LIN {X 0,Y 523.933,Z 425.84,A -85,B 0,C 180,E1 -4843.639,E2 -4843.639} C_VEL
LIN {X 0,Y 523.933,Z 425.846,A -85,B 0,C 180,E1 -4846.028,E2 -4846.028} C_VEL
LIN {X 0,Y 524.007,Z 425.841,A -85,B 0,C 180,E1 -4848.394,E2 -4848.394} C_VEL
LIN {X 0,Y 524,Z 425.833,A -85,B 0,C 180,E1 -4851.516,E2 -4851.516} C_VEL
LIN {X 0,Y 524.077,Z 425.829,A -85,B 0,C 180,E1 -4854.614,E2 -4854.614} C_VEL
LIN {X 0,Y 524.106,Z 425.82,A -85,B 0,C 180,E1 -4857.695,E2 -4857.695} C_VEL
LIN {X 0,Y 524.118,Z 425.82,A -85,B 0,C 180,E1 -4860.769,E2 -4860.769} C_VEL
LIN {X 0,Y 524.069,Z 425.826,A -85,B 0,C 180,E1 -4863.075,E2 -4863.075} C_VEL
LIN {X 0,Y 524.045,Z 425.833,A -85,B 0,C 180,E1 -4866.159,E2 -4866.159} C_VEL
LIN {X 0,Y 523.996,Z 425.834,A -85,B 0,C 180,E1 -4869.262,E2 -4869.262} C_VEL
LIN {X 0,Y 523.996,Z 425.834,A -85,B 0,C 180,E1 -4871.74,E2 -4871.74} C_VEL
LIN {X 0,Y 523.987,Z 425.837,A -85,B 0,C 180,E1 -4875.053,E2 -4875.053} C_VEL
LIN {X 0,Y 523.958,Z 425.842,A -85,B 0,C 180,E1 -4877.969,E2 -4877.969} C_VEL
LIN {X 0,Y 523.966,Z 425.847,A -85,B 0,C 180,E1 -4880.411,E2 -4880.411} C_VEL
LIN {X 0,Y 523.911,Z 425.848,A -85,B 0,C 180,E1 -4882.894,E2 -4882.894} C_VEL
LIN {X 0,Y 523.949,Z 425.841,A -85,B 0,C 180,E1 -4885.419,E2 -4885.419} C_VEL
LIN {X 0,Y 523.966,Z 425.842,A -85,B 0,C 180,E1 -4887.999,E2 -4887.999} C_VEL
LIN {X 0,Y 523.948,Z 425.845,A -85,B 0,C 180,E1 -4890.857,E2 -4890.857} C_VEL
LIN {X 0,Y 523.958,Z 425.841,A -85,B 0,C 180,E1 -4893.736,E2 -4893.736} C_VEL
LIN {X 0,Y 523.921,Z 425.852,A -85,B 0,C 180,E1 -4896.406,E2 -4896.406} C_VEL
LIN {X 0,Y 523.956,Z 425.844,A -85,B 0,C 180,E1 -4899.082,E2 -4899.082} C_VEL
LIN {X 0,Y 523.953,Z 425.847,A -85,B 0,C 180,E1 -4902.119,E2 -4902.119} C_VEL
LIN {X 0,Y 524.002,Z 426.023,A -85,B 0,C 180,E1 -4903.252,E2 -4903.252} C_VEL
LIN {X 0,Y 525.992,Z 435.927,A -85,B 0,C 180,E1 -4904.916,E2 -4904.916} C_VEL
LIN {X 0,Y 525.874,Z 439.256,A -85,B 0,C 180,E1 -4905.427,E2 -4905.427} C_VEL
LIN {X 0,Y 525.617,Z 441.85,A -85,B 0,C 180,E1 -4905.741,E2 -4905.741} C_VEL
LIN {X 0,Y 524.85,Z 446.612,A -85,B 0,C 180,E1 -4906.106,E2 -4906.106} C_VEL
LIN {X 0,Y 523.874,Z 451.969,A -85,B 0,C 180,E1 -4906.359,E2 -4906.359} C_VEL
LIN {X 0,Y 522.61,Z 459.806,A -85,B 0,C 180,E1 -4906.576,E2 -4906.576} C_VEL
LIN {X 0,Y 521.99,Z 467.878,A -85,B 0,C 180,E1 -4906.711,E2 -4906.711} C_VEL
LIN {X 0,Y 520.915,Z 611.533,A -85,B 0,C 180,E1 -4908.76,E2 -4908.76} C_VEL
LIN {X 0,Y 520.597,Z 626.808,A -85,B 0,C 180,E1 -4909.129,E2 -4909.129} C_VEL
LIN {X 0,Y 520.217,Z 641.341,A -85,B 0,C 180,E1 -4909.639,E2 -4909.639} C_VEL
LIN {X 0,Y 519.75,Z 655.45,A -85,B 0,C 180,E1 -4910.291,E2 -4910.291} C_VEL
LIN {X 0,Y 519.293,Z 667.726,A -85,B 0,C 180,E1 -4911.001,E2 -4911.001} C_VEL
LIN {X 0,Y 518.8,Z 680.193,A -85,B 0,C 180,E1 -4911.873,E2 -4911.873} C_VEL
LIN {X 0,Y 518.29,Z 692.73,A -85,B 0,C 180,E1 -4912.931,E2 -4912.931} C_VEL
LIN {X 0,Y 517.723,Z 704.894,A -85,B 0,C 180,E1 -4914.169,E2 -4914.169} C_VEL
LIN {X 0,Y 517.327,Z 715.213,A -85,B 0,C 180,E1 -4915.43,E2 -4915.43} C_VEL
LIN {X 0,Y 516.961,Z 724.771,A -85,B 0,C 180,E1 -4916.826,E2 -4916.826} C_VEL
LIN {X 0,Y 516.71,Z 732.578,A -85,B 0,C 180,E1 -4918.194,E2 -4918.194} C_VEL
LIN {X 0,Y 516.51,Z 739.956,A -85,B 0,C 180,E1 -4919.773,E2 -4919.773} C_VEL
LIN {X 0,Y 516.361,Z 745.035,A -85,B 0,C 180,E1 -4921.108,E2 -4921.108} C_VEL
LIN {X 0,Y 516.279,Z 750.189,A -85,B 0,C 180,E1 -4922.87,E2 -4922.87} C_VEL
LIN {X 0,Y 516.196,Z 752.938,A -85,B 0,C 180,E1 -4924.172,E2 -4924.172} C_VEL
LIN {X 0,Y 516.177,Z 755.377,A -85,B 0,C 180,E1 -4925.892,E2 -4925.892} C_VEL
LIN {X 0,Y 516.144,Z 756.413,A -85,B 0,C 180,E1 -4927.589,E2 -4927.589} C_VEL
LIN {X 0,Y 516.172,Z 756.115,A -85,B 0,C 180,E1 -4929.268,E2 -4929.268} C_VEL
LIN {X 0,Y 516.166,Z 754.527,A -85,B 0,C 180,E1 -4930.927,E2 -4930.927} C_VEL
LIN {X 0,Y 516.24,Z 751.657,A -85,B 0,C 180,E1 -4932.573,E2 -4932.573} C_VEL
LIN {X 0,Y 516.346,Z 747.496,A -85,B 0,C 180,E1 -4934.204,E2 -4934.204} C_VEL
LIN {X 0,Y 516.472,Z 741.966,A -85,B 0,C 180,E1 -4935.822,E2 -4935.822} C_VEL
LIN {X 0,Y 516.605,Z 734.953,A -85,B 0,C 180,E1 -4937.429,E2 -4937.429} C_VEL
LIN {X 0,Y 516.88,Z 727.372,A -85,B 0,C 180,E1 -4938.841,E2 -4938.841} C_VEL
LIN {X 0,Y 517.18,Z 718.444,A -85,B 0,C 180,E1 -4940.221,E2 -4940.221} C_VEL
LIN {X 0,Y 517.658,Z 707.481,A -85,B 0,C 180,E1 -4941.628,E2 -4941.628} C_VEL
LIN {X 0,Y 518.13,Z 696.22,A -85,B 0,C 180,E1 -4942.83,E2 -4942.83} C_VEL
LIN {X 0,Y 518.663,Z 683.329,A -85,B 0,C 180,E1 -4943.973,E2 -4943.973} C_VEL
LIN {X 0,Y 519.217,Z 669.849,A -85,B 0,C 180,E1 -4944.953,E2 -4944.953} C_VEL
LIN {X 0,Y 519.691,Z 656.693,A -85,B 0,C 180,E1 -4945.735,E2 -4945.735} C_VEL
LIN {X 0,Y 520.165,Z 642.175,A -85,B 0,C 180,E1 -4946.418,E2 -4946.418} C_VEL
LIN {X 0,Y 520.611,Z 627.046,A -85,B 0,C 180,E1 -4946.952,E2 -4946.952} C_VEL
LIN {X 0,Y 520.884,Z 611.84,A -85,B 0,C 180,E1 -4947.325,E2 -4947.325} C_VEL
LIN {X 0,Y 521.976,Z 460.856,A -85,B 0,C 180,E1 -4949.481,E2 -4949.481} C_VEL
LIN {X 0,Y 518.847,Z 446.809,A -85,B 0,C 180,E1 -4949.826,E2 -4949.826} C_VEL
LIN {X 0,Y 519.1,Z 436.953,A -85,B 0,C 180,E1 -4951.358,E2 -4951.358} C_VEL
LIN {X 0,Y 517.017,Z 426.712,A -85,B 0,C 180,E1 -4953.117,E2 -4953.117} C_VEL
LIN {X 0,Y 516.993,Z 426.711,A -85,B 0,C 180,E1 -4956.244,E2 -4956.244} C_VEL
LIN {X 0,Y 516.973,Z 426.711,A -85,B 0,C 180,E1 -4958.601,E2 -4958.601} C_VEL
LIN {X 0,Y 516.989,Z 426.715,A -85,B 0,C 180,E1 -4961.824,E2 -4961.824} C_VEL
LIN {X 0,Y 516.949,Z 426.715,A -85,B 0,C 180,E1 -4965.147,E2 -4965.147} C_VEL
LIN {X 0,Y 516.929,Z 426.716,A -85,B 0,C 180,E1 -4968.222,E2 -4968.222} C_VEL
LIN {X 0,Y 516.917,Z 426.716,A -85,B 0,C 180,E1 -4970.701,E2 -4970.701} C_VEL
LIN {X 0,Y 516.916,Z 426.717,A -85,B 0,C 180,E1 -4974.072,E2 -4974.072} C_VEL
LIN {X 0,Y 516.93,Z 426.714,A -85,B 0,C 180,E1 -4976.658,E2 -4976.658} C_VEL
LIN {X 0,Y 516.915,Z 426.721,A -85,B 0,C 180,E1 -4979.524,E2 -4979.524} C_VEL
LIN {X 0,Y 516.904,Z 426.713,A -85,B 0,C 180,E1 -4982.544,E2 -4982.544} C_VEL
LIN {X 0,Y 516.884,Z 426.725,A -85,B 0,C 180,E1 -4985.332,E2 -4985.332} C_VEL
LIN {X 0,Y 516.885,Z 426.721,A -85,B 0,C 180,E1 -4987.943,E2 -4987.943} C_VEL
LIN {X 0,Y 516.889,Z 426.719,A -85,B 0,C 180,E1 -4990.741,E2 -4990.741} C_VEL
LIN {X 0,Y 516.907,Z 426.715,A -85,B 0,C 180,E1 -4992.829,E2 -4992.829} C_VEL
LIN {X 0,Y 516.925,Z 426.715,A -85,B 0,C 180,E1 -4995.01,E2 -4995.01} C_VEL
LIN {X 0,Y 516.924,Z 426.712,A -85,B 0,C 180,E1 -4998.397,E2 -4998.397} C_VEL
LIN {X 0,Y 516.888,Z 426.723,A -85,B 0,C 180,E1 -5001.284,E2 -5001.284} C_VEL
LIN {X 0,Y 516.894,Z 426.717,A -85,B 0,C 180,E1 -5004.221,E2 -5004.221} C_VEL
LIN {X 0,Y 516.898,Z 426.719,A -85,B 0,C 180,E1 -5007.053,E2 -5007.053} C_VEL
LIN {X 0,Y 516.893,Z 426.721,A -85,B 0,C 180,E1 -5009.796,E2 -5009.796} C_VEL
LIN {X 0,Y 516.932,Z 426.714,A -85,B 0,C 180,E1 -5012.467,E2 -5012.467} C_VEL
LIN {X 0,Y 516.911,Z 426.717,A -85,B 0,C 180,E1 -5015.072,E2 -5015.072} C_VEL
LIN {X 0,Y 516.886,Z 426.719,A -85,B 0,C 180,E1 -5018.462,E2 -5018.462} C_VEL
LIN {X 0,Y 516.904,Z 426.718,A -85,B 0,C 180,E1 -5020.955,E2 -5020.955} C_VEL
LIN {X 0,Y 516.915,Z 426.717,A -85,B 0,C 180,E1 -5023.41,E2 -5023.41} C_VEL
LIN {X 0,Y 516.896,Z 426.725,A -85,B 0,C 180,E1 -5025.833,E2 -5025.833} C_VEL
LIN {X 0,Y 516.966,Z 426.709,A -85,B 0,C 180,E1 -5028.233,E2 -5028.233} C_VEL
LIN {X 0,Y 516.97,Z 426.709,A -85,B 0,C 180,E1 -5031.399,E2 -5031.399} C_VEL
LIN {X 0,Y 517.01,Z 426.712,A -85,B 0,C 180,E1 -5033.757,E2 -5033.757} C_VEL
LIN {X 0,Y 517.083,Z 426.698,A -85,B 0,C 180,E1 -5037.663,E2 -5037.663} C_VEL
LIN {X 0,Y 517.094,Z 426.694,A -85,B 0,C 180,E1 -5040.779,E2 -5040.779} C_VEL
LIN {X 0,Y 517.014,Z 426.703,A -85,B 0,C 180,E1 -5043.117,E2 -5043.117} C_VEL
LIN {X 0,Y 517.009,Z 426.704,A -85,B 0,C 180,E1 -5046.243,E2 -5046.243} C_VEL
LIN {X 0,Y 516.953,Z 426.716,A -85,B 0,C 180,E1 -5049.389,E2 -5049.389} C_VEL
LIN {X 0,Y 516.951,Z 426.712,A -85,B 0,C 180,E1 -5051.807,E2 -5051.807} C_VEL
LIN {X 0,Y 516.943,Z 426.714,A -85,B 0,C 180,E1 -5055.146,E2 -5055.146} C_VEL
LIN {X 0,Y 516.924,Z 426.711,A -85,B 0,C 180,E1 -5058.222,E2 -5058.222} C_VEL
LIN {X 0,Y 516.912,Z 426.716,A -85,B 0,C 180,E1 -5060.701,E2 -5060.701} C_VEL
LIN {X 0,Y 516.911,Z 426.72,A -85,B 0,C 180,E1 -5064.072,E2 -5064.072} C_VEL
LIN {X 0,Y 516.926,Z 426.714,A -85,B 0,C 180,E1 -5066.658,E2 -5066.658} C_VEL
LIN {X 0,Y 516.91,Z 426.722,A -85,B 0,C 180,E1 -5069.524,E2 -5069.524} C_VEL
LIN {X 0,Y 516.897,Z 426.718,A -85,B 0,C 180,E1 -5072.544,E2 -5072.544} C_VEL
LIN {X 0,Y 516.883,Z 426.724,A -85,B 0,C 180,E1 -5075.332,E2 -5075.332} C_VEL
LIN {X 0,Y 516.881,Z 426.726,A -85,B 0,C 180,E1 -5077.943,E2 -5077.943} C_VEL
LIN {X 0,Y 516.884,Z 426.72,A -85,B 0,C 180,E1 -5080.742,E2 -5080.742} C_VEL
LIN {X 0,Y 516.883,Z 426.72,A -85,B 0,C 180,E1 -5082.831,E2 -5082.831} C_VEL
LIN {X 0,Y 516.923,Z 426.716,A -85,B 0,C 180,E1 -5085.01,E2 -5085.01} C_VEL
LIN {X 0,Y 516.916,Z 426.718,A -85,B 0,C 180,E1 -5088.398,E2 -5088.398} C_VEL
LIN {X 0,Y 516.881,Z 426.724,A -85,B 0,C 180,E1 -5091.284,E2 -5091.284} C_VEL
LIN {X 0,Y 516.871,Z 426.727,A -85,B 0,C 180,E1 -5094.22,E2 -5094.22} C_VEL
LIN {X 0,Y 516.895,Z 426.723,A -85,B 0,C 180,E1 -5097.053,E2 -5097.053} C_VEL
LIN {X 0,Y 516.893,Z 426.728,A -85,B 0,C 180,E1 -5099.796,E2 -5099.796} C_VEL
LIN {X 0,Y 516.935,Z 426.735,A -85,B 0,C 180,E1 -5101.653,E2 -5101.653} C_VEL
LIN {X 0,Y 520.07,Z 440.507,A -85,B 0,C 180,E1 -5103.732,E2 -5103.732} C_VEL
LIN {X 0,Y 519.386,Z 460.989,A -85,B 0,C 180,E1 -5106.473,E2 -5106.473} C_VEL
LIN {X 0,Y 518.966,Z 474.064,A -85,B 0,C 180,E1 -5108.202,E2 -5108.202} C_VEL
LIN {X 0,Y 521.939,Z 489.827,A -85,B 0,C 180,E1 -5108.57,E2 -5108.57} C_VEL
LIN {X 0,Y 520.844,Z 639.891,A -85,B 0,C 180,E1 -5110.705,E2 -5110.705} C_VEL
LIN {X 0,Y 520.532,Z 655.089,A -85,B 0,C 180,E1 -5111.067,E2 -5111.067} C_VEL
LIN {X 0,Y 520.144,Z 670.136,A -85,B 0,C 180,E1 -5111.589,E2 -5111.589} C_VEL
LIN {X 0,Y 519.687,Z 683.207,A -85,B 0,C 180,E1 -5112.183,E2 -5112.183} C_VEL
LIN {X 0,Y 519.207,Z 697.158,A -85,B 0,C 180,E1 -5112.979,E2 -5112.979} C_VEL
LIN {X 0,Y 518.693,Z 710.453,A -85,B 0,C 180,E1 -5113.913,E2 -5113.913} C_VEL
LIN {X 0,Y 518.16,Z 721.964,A -85,B 0,C 180,E1 -5114.882,E2 -5114.882} C_VEL
LIN {X 0,Y 517.701,Z 733.666,A -85,B 0,C 180,E1 -5116.056,E2 -5116.056} C_VEL
LIN {X 0,Y 517.313,Z 743.673,A -85,B 0,C 180,E1 -5117.246,E2 -5117.246} C_VEL
LIN {X 0,Y 516.972,Z 753.465,A -85,B 0,C 180,E1 -5118.631,E2 -5118.631} C_VEL
LIN {X 0,Y 516.68,Z 761.63,A -85,B 0,C 180,E1 -5120.012,E2 -5120.012} C_VEL
LIN {X 0,Y 516.541,Z 768.382,A -85,B 0,C 180,E1 -5121.392,E2 -5121.392} C_VEL
LIN {X 0,Y 516.391,Z 774.604,A -85,B 0,C 180,E1 -5122.964,E2 -5122.964} C_VEL
LIN {X 0,Y 516.373,Z 779.384,A -85,B 0,C 180,E1 -5124.533,E2 -5124.533} C_VEL
LIN {X 0,Y 516.307,Z 782.885,A -85,B 0,C 180,E1 -5126.097,E2 -5126.097} C_VEL
LIN {X 0,Y 516.257,Z 785.188,A -85,B 0,C 180,E1 -5127.659,E2 -5127.659} C_VEL
LIN {X 0,Y 516.157,Z 786.347,A -85,B 0,C 180,E1 -5129.219,E2 -5129.219} C_VEL
LIN {X 0,Y 516.157,Z 786.346,A -85,B 0,C 180,E1 -5130.78,E2 -5130.78} C_VEL
LIN {X 0,Y 516.257,Z 785.185,A -85,B 0,C 180,E1 -5132.34,E2 -5132.34} C_VEL
LIN {X 0,Y 516.307,Z 782.882,A -85,B 0,C 180,E1 -5133.902,E2 -5133.902} C_VEL
LIN {X 0,Y 516.372,Z 779.388,A -85,B 0,C 180,E1 -5135.466,E2 -5135.466} C_VEL
LIN {X 0,Y 516.391,Z 774.611,A -85,B 0,C 180,E1 -5137.035,E2 -5137.035} C_VEL
LIN {X 0,Y 516.54,Z 768.382,A -85,B 0,C 180,E1 -5138.607,E2 -5138.607} C_VEL
LIN {X 0,Y 516.756,Z 760.538,A -85,B 0,C 180,E1 -5140.183,E2 -5140.183} C_VEL
LIN {X 0,Y 516.999,Z 752.194,A -85,B 0,C 180,E1 -5141.566,E2 -5141.566} C_VEL
LIN {X 0,Y 517.382,Z 742.143,A -85,B 0,C 180,E1 -5142.951,E2 -5142.951} C_VEL
LIN {X 0,Y 517.775,Z 731.862,A -85,B 0,C 180,E1 -5144.141,E2 -5144.141} C_VEL
LIN {X 0,Y 518.277,Z 719.898,A -85,B 0,C 180,E1 -5145.306,E2 -5145.306} C_VEL
LIN {X 0,Y 518.78,Z 707.325,A -85,B 0,C 180,E1 -5146.325,E2 -5146.325} C_VEL
LIN {X 0,Y 519.332,Z 693.947,A -85,B 0,C 180,E1 -5147.219,E2 -5147.219} C_VEL
LIN {X 0,Y 519.834,Z 679.183,A -85,B 0,C 180,E1 -5148.014,E2 -5148.014} C_VEL
LIN {X 0,Y 520.267,Z 664.898,A -85,B 0,C 180,E1 -5148.61,E2 -5148.61} C_VEL
LIN {X 0,Y 520.638,Z 650,A -85,B 0,C 180,E1 -5149.069,E2 -5149.069} C_VEL
LIN {X 0,Y 520.902,Z 635.089,A -85,B 0,C 180,E1 -5149.373,E2 -5149.373} C_VEL
LIN {X 0,Y 521.915,Z 489.347,A -85,B 0,C 180,E1 -5151.437,E2 -5151.437} C_VEL
LIN {X 0,Y 518.938,Z 473.889,A -85,B 0,C 180,E1 -5151.806,E2 -5151.806} C_VEL
LIN {X 0,Y 519.69,Z 451.385,A -85,B 0,C 180,E1 -5154.785,E2 -5154.785} C_VEL
LIN {X 0,Y 520.017,Z 440.332,A -85,B 0,C 180,E1 -5156.27,E2 -5156.27} C_VEL
LIN {X 0,Y 516.932,Z 426.726,A -85,B 0,C 180,E1 -5158.346,E2 -5158.346} C_VEL
LIN {X 0,Y 516.889,Z 426.723,A -85,B 0,C 180,E1 -5161.109,E2 -5161.109} C_VEL
LIN {X 0,Y 516.908,Z 426.722,A -85,B 0,C 180,E1 -5163.966,E2 -5163.966} C_VEL
LIN {X 0,Y 516.879,Z 426.724,A -85,B 0,C 180,E1 -5166.745,E2 -5166.745} C_VEL
LIN {X 0,Y 516.907,Z 426.72,A -85,B 0,C 180,E1 -5169.718,E2 -5169.718} C_VEL
LIN {X 0,Y 516.9,Z 426.719,A -85,B 0,C 180,E1 -5172.828,E2 -5172.828} C_VEL
LIN {X 0,Y 516.917,Z 426.718,A -85,B 0,C 180,E1 -5175.01,E2 -5175.01} C_VEL
LIN {X 0,Y 516.911,Z 426.725,A -85,B 0,C 180,E1 -5178.398,E2 -5178.398} C_VEL
LIN {X 0,Y 516.877,Z 426.721,A -85,B 0,C 180,E1 -5181.284,E2 -5181.284} C_VEL
LIN {X 0,Y 516.885,Z 426.727,A -85,B 0,C 180,E1 -5184.221,E2 -5184.221} C_VEL
LIN {X 0,Y 516.892,Z 426.718,A -85,B 0,C 180,E1 -5187.053,E2 -5187.053} C_VEL
LIN {X 0,Y 516.885,Z 426.721,A -85,B 0,C 180,E1 -5189.796,E2 -5189.796} C_VEL
LIN {X 0,Y 516.923,Z 426.72,A -85,B 0,C 180,E1 -5192.467,E2 -5192.467} C_VEL
LIN {X 0,Y 516.905,Z 426.718,A -85,B 0,C 180,E1 -5195.072,E2 -5195.072} C_VEL
LIN {X 0,Y 516.88,Z 426.726,A -85,B 0,C 180,E1 -5198.462,E2 -5198.462} C_VEL
LIN {X 0,Y 516.898,Z 426.72,A -85,B 0,C 180,E1 -5200.955,E2 -5200.955} C_VEL
LIN {X 0,Y 516.909,Z 426.714,A -85,B 0,C 180,E1 -5203.41,E2 -5203.41} C_VEL
LIN {X 0,Y 516.888,Z 426.722,A -85,B 0,C 180,E1 -5205.834,E2 -5205.834} C_VEL
LIN {X 0,Y 516.996,Z 426.712,A -85,B 0,C 180,E1 -5208.235,E2 -5208.235} C_VEL
LIN {X 0,Y 516.965,Z 426.709,A -85,B 0,C 180,E1 -5211.4,E2 -5211.4} C_VEL
LIN {X 0,Y 517.003,Z 426.706,A -85,B 0,C 180,E1 -5213.757,E2 -5213.757} C_VEL
LIN {X 0,Y 517.078,Z 426.695,A -85,B 0,C 180,E1 -5217.663,E2 -5217.663} C_VEL
LIN {X 0,Y 517.088,Z 426.695,A -85,B 0,C 180,E1 -5220.779,E2 -5220.779} C_VEL
LIN {X 0,Y 517.01,Z 426.705,A -85,B 0,C 180,E1 -5223.117,E2 -5223.117} C_VEL
LIN {X 0,Y 517.008,Z 426.711,A -85,B 0,C 180,E1 -5226.243,E2 -5226.243} C_VEL
LIN {X 0,Y 516.95,Z 426.712,A -85,B 0,C 180,E1 -5229.39,E2 -5229.39} C_VEL
LIN {X 0,Y 516.945,Z 426.713,A -85,B 0,C 180,E1 -5231.808,E2 -5231.808} C_VEL
LIN {X 0,Y 516.94,Z 426.714,A -85,B 0,C 180,E1 -5235.148,E2 -5235.148} C_VEL
LIN {X 0,Y 516.92,Z 426.722,A -85,B 0,C 180,E1 -5238.223,E2 -5238.223} C_VEL
LIN {X 0,Y 516.907,Z 426.722,A -85,B 0,C 180,E1 -5240.702,E2 -5240.702} C_VEL
LIN {X 0,Y 516.905,Z 426.722,A -85,B 0,C 180,E1 -5244.073,E2 -5244.073} C_VEL
LIN {X 0,Y 516.924,Z 426.72,A -85,B 0,C 180,E1 -5246.658,E2 -5246.658} C_VEL
LIN {X 0,Y 516.92,Z 426.716,A -85,B 0,C 180,E1 -5249.527,E2 -5249.527} C_VEL
LIN {X 0,Y 516.897,Z 426.724,A -85,B 0,C 180,E1 -5252.545,E2 -5252.545} C_VEL
LIN {X 0,Y 516.88,Z 426.723,A -85,B 0,C 180,E1 -5255.333,E2 -5255.333} C_VEL
LIN {X 0,Y 516.878,Z 426.726,A -85,B 0,C 180,E1 -5257.944,E2 -5257.944} C_VEL
LIN {X 0,Y 516.901,Z 426.725,A -85,B 0,C 180,E1 -5260.74,E2 -5260.74} C_VEL
LIN {X 0,Y 516.934,Z 426.875,A -85,B 0,C 180,E1 -5262.993,E2 -5262.993} C_VEL
LIN {X 0,Y 519.112,Z 437.159,A -85,B 0,C 180,E1 -5264.749,E2 -5264.749} C_VEL
LIN {X 0,Y 518.838,Z 446.855,A -85,B 0,C 180,E1 -5266.255,E2 -5266.255} C_VEL
LIN {X 0,Y 521.986,Z 460.996,A -85,B 0,C 180,E1 -5266.61,E2 -5266.61} C_VEL
LIN {X 0,Y 521.99,Z 467.878,A -85,B 0,C 180,E1 -5266.711,E2 -5266.711} C_VEL
LIN {X 0,Y 521.333,Z 473.722,A -85,B 0,C 180,E1 -5266.768,E2 -5266.768} C_VEL
LIN {X 0,Y 515.846,Z 492.777,A -85,B 0,C 180,E1 -5266.809,E2 -5266.809} C_VEL
LIN {X 0,Y 515.068,Z 498.627,A -85,B 0,C 180,E1 -5266.861,E2 -5266.861} C_VEL
LIN {X 0,Y 514.235,Z 611.582,A -85,B 0,C 180,E1 -5268.498,E2 -5268.498} C_VEL
LIN {X 0,Y 513.886,Z 626.632,A -85,B 0,C 180,E1 -5268.863,E2 -5268.863} C_VEL
LIN {X 0,Y 513.473,Z 641.413,A -85,B 0,C 180,E1 -5269.384,E2 -5269.384} C_VEL
LIN {X 0,Y 513.002,Z 654.957,A -85,B 0,C 180,E1 -5270.015,E2 -5270.015} C_VEL
LIN {X 0,Y 512.503,Z 667.867,A -85,B 0,C 180,E1 -5270.766,E2 -5270.766} C_VEL
LIN {X 0,Y 511.934,Z 680.463,A -85,B 0,C 180,E1 -5271.656,E2 -5271.656} C_VEL
LIN {X 0,Y 511.422,Z 692.408,A -85,B 0,C 180,E1 -5272.674,E2 -5272.674} C_VEL
LIN {X 0,Y 510.82,Z 704.352,A -85,B 0,C 180,E1 -5273.893,E2 -5273.893} C_VEL
LIN {X 0,Y 510.405,Z 714.649,A -85,B 0,C 180,E1 -5275.151,E2 -5275.151} C_VEL
LIN {X 0,Y 509.973,Z 724.235,A -85,B 0,C 180,E1 -5276.549,E2 -5276.549} C_VEL
LIN {X 0,Y 509.679,Z 732.182,A -85,B 0,C 180,E1 -5277.936,E2 -5277.936} C_VEL
LIN {X 0,Y 509.474,Z 738.715,A -85,B 0,C 180,E1 -5279.31,E2 -5279.31} C_VEL
LIN {X 0,Y 509.318,Z 744.305,A -85,B 0,C 180,E1 -5280.747,E2 -5280.747} C_VEL
LIN {X 0,Y 509.213,Z 749.551,A -85,B 0,C 180,E1 -5282.474,E2 -5282.474} C_VEL
LIN {X 0,Y 509.104,Z 752.578,A -85,B 0,C 180,E1 -5283.806,E2 -5283.806} C_VEL
LIN {X 0,Y 509.08,Z 755.231,A -85,B 0,C 180,E1 -5285.534,E2 -5285.534} C_VEL
LIN {X 0,Y 509.038,Z 756.521,A -85,B 0,C 180,E1 -5287.259,E2 -5287.259} C_VEL
LIN {X 0,Y 509.061,Z 756.479,A -85,B 0,C 180,E1 -5288.965,E2 -5288.965} C_VEL
LIN {X 0,Y 509.096,Z 755.136,A -85,B 0,C 180,E1 -5290.652,E2 -5290.652} C_VEL
LIN {X 0,Y 509.135,Z 752.508,A -85,B 0,C 180,E1 -5292.322,E2 -5292.322} C_VEL
LIN {X 0,Y 509.254,Z 748.579,A -85,B 0,C 180,E1 -5293.978,E2 -5293.978} C_VEL
LIN {X 0,Y 509.362,Z 744.437,A -85,B 0,C 180,E1 -5295.301,E2 -5295.301} C_VEL
LIN {X 0,Y 509.479,Z 738.415,A -85,B 0,C 180,E1 -5296.844,E2 -5296.844} C_VEL
LIN {X 0,Y 509.719,Z 731.814,A -85,B 0,C 180,E1 -5298.224,E2 -5298.224} C_VEL
LIN {X 0,Y 510.002,Z 723.366,A -85,B 0,C 180,E1 -5299.681,E2 -5299.681} C_VEL
LIN {X 0,Y 510.415,Z 713.525,A -85,B 0,C 180,E1 -5301.089,E2 -5301.089} C_VEL
LIN {X 0,Y 510.965,Z 701.852,A -85,B 0,C 180,E1 -5302.472,E2 -5302.472} C_VEL
LIN {X 0,Y 511.535,Z 689.383,A -85,B 0,C 180,E1 -5303.69,E2 -5303.69} C_VEL
LIN {X 0,Y 512.081,Z 677.163,A -85,B 0,C 180,E1 -5304.685,E2 -5304.685} C_VEL
LIN {X 0,Y 512.694,Z 663.81,A -85,B 0,C 180,E1 -5305.578,E2 -5305.578} C_VEL
LIN {X 0,Y 513.191,Z 650.074,A -85,B 0,C 180,E1 -5306.32,E2 -5306.32} C_VEL
LIN {X 0,Y 513.673,Z 634.94,A -85,B 0,C 180,E1 -5306.953,E2 -5306.953} C_VEL
LIN {X 0,Y 514.043,Z 619.208,A -85,B 0,C 180,E1 -5307.427,E2 -5307.427} C_VEL
LIN {X 0,Y 514.26,Z 603.725,A -85,B 0,C 180,E1 -5307.724,E2 -5307.724} C_VEL
LIN {X 0,Y 515.276,Z 461.394,A -85,B 0,C 180,E1 -5309.769,E2 -5309.769} C_VEL
LIN {X 0,Y 512.043,Z 446.867,A -85,B 0,C 180,E1 -5310.153,E2 -5310.153} C_VEL
LIN {X 0,Y 512.271,Z 439.079,A -85,B 0,C 180,E1 -5311.376,E2 -5311.376} C_VEL
LIN {X 0,Y 510.494,Z 429.788,A -85,B 0,C 180,E1 -5312.96,E2 -5312.96} C_VEL
LIN {X 0,Y 509.929,Z 427.595,A -85,B 0,C 180,E1 -5313.358,E2 -5313.358} C_VEL
LIN {X 0,Y 509.941,Z 427.589,A -85,B 0,C 180,E1 -5316.33,E2 -5316.33} C_VEL
LIN {X 0,Y 509.919,Z 427.59,A -85,B 0,C 180,E1 -5318.72,E2 -5318.72} C_VEL
LIN {X 0,Y 509.956,Z 427.59,A -85,B 0,C 180,E1 -5321.931,E2 -5321.931} C_VEL
LIN {X 0,Y 509.899,Z 427.595,A -85,B 0,C 180,E1 -5325.242,E2 -5325.242} C_VEL
LIN {X 0,Y 509.886,Z 427.596,A -85,B 0,C 180,E1 -5327.999,E2 -5327.999} C_VEL
LIN {X 0,Y 509.855,Z 427.597,A -85,B 0,C 180,E1 -5331.002,E2 -5331.002} C_VEL
LIN {X 0,Y 509.841,Z 427.605,A -85,B 0,C 180,E1 -5333.563,E2 -5333.563} C_VEL
LIN {X 0,Y 509.916,Z 427.589,A -85,B 0,C 180,E1 -5336.379,E2 -5336.379} C_VEL
LIN {X 0,Y 509.881,Z 427.59,A -85,B 0,C 180,E1 -5338.844,E2 -5338.844} C_VEL
LIN {X 0,Y 509.83,Z 427.605,A -85,B 0,C 180,E1 -5341.59,E2 -5341.59} C_VEL
LIN {X 0,Y 509.856,Z 427.596,A -85,B 0,C 180,E1 -5344.413,E2 -5344.413} C_VEL
LIN {X 0,Y 509.822,Z 427.603,A -85,B 0,C 180,E1 -5347.34,E2 -5347.34} C_VEL
LIN {X 0,Y 509.842,Z 427.598,A -85,B 0,C 180,E1 -5350.382,E2 -5350.382} C_VEL
LIN {X 0,Y 509.842,Z 427.596,A -85,B 0,C 180,E1 -5353.064,E2 -5353.064} C_VEL
LIN {X 0,Y 509.834,Z 427.605,A -85,B 0,C 180,E1 -5355.792,E2 -5355.792} C_VEL
LIN {X 0,Y 509.867,Z 427.59,A -85,B 0,C 180,E1 -5358.575,E2 -5358.575} C_VEL
LIN {X 0,Y 509.854,Z 427.602,A -85,B 0,C 180,E1 -5361.786,E2 -5361.786} C_VEL
LIN {X 0,Y 509.848,Z 427.593,A -85,B 0,C 180,E1 -5364.623,E2 -5364.623} C_VEL
LIN {X 0,Y 509.864,Z 427.601,A -85,B 0,C 180,E1 -5367.481,E2 -5367.481} C_VEL
LIN {X 0,Y 509.859,Z 427.592,A -85,B 0,C 180,E1 -5370.273,E2 -5370.273} C_VEL
LIN {X 0,Y 509.889,Z 427.592,A -85,B 0,C 180,E1 -5372.944,E2 -5372.944} C_VEL
LIN {X 0,Y 509.866,Z 427.599,A -85,B 0,C 180,E1 -5375.574,E2 -5375.574} C_VEL
LIN {X 0,Y 509.851,Z 427.596,A -85,B 0,C 180,E1 -5378.998,E2 -5378.998} C_VEL
LIN {X 0,Y 509.889,Z 427.591,A -85,B 0,C 180,E1 -5381.999,E2 -5381.999} C_VEL
LIN {X 0,Y 509.911,Z 427.585,A -85,B 0,C 180,E1 -5384.819,E2 -5384.819} C_VEL
LIN {X 0,Y 509.901,Z 427.59,A -85,B 0,C 180,E1 -5388.124,E2 -5388.124} C_VEL
LIN {X 0,Y 509.916,Z 427.586,A -85,B 0,C 180,E1 -5391.28,E2 -5391.28} C_VEL
LIN {X 0,Y 509.978,Z 427.589,A -85,B 0,C 180,E1 -5393.67,E2 -5393.67} C_VEL
LIN {X 0,Y 510.054,Z 427.572,A -85,B 0,C 180,E1 -5397.631,E2 -5397.631} C_VEL
LIN {X 0,Y 510.064,Z 427.569,A -85,B 0,C 180,E1 -5400.789,E2 -5400.789} C_VEL
LIN {X 0,Y 509.956,Z 427.582,A -85,B 0,C 180,E1 -5403.16,E2 -5403.16} C_VEL
LIN {X 0,Y 509.978,Z 427.579,A -85,B 0,C 180,E1 -5406.329,E2 -5406.329} C_VEL
LIN {X 0,Y 509.916,Z 427.588,A -85,B 0,C 180,E1 -5408.72,E2 -5408.72} C_VEL
LIN {X 0,Y 509.904,Z 427.589,A -85,B 0,C 180,E1 -5411.931,E2 -5411.931} C_VEL
LIN {X 0,Y 509.893,Z 427.593,A -85,B 0,C 180,E1 -5415.242,E2 -5415.242} C_VEL
LIN {X 0,Y 509.888,Z 427.59,A -85,B 0,C 180,E1 -5418.001,E2 -5418.001} C_VEL
LIN {X 0,Y 509.85,Z 427.596,A -85,B 0,C 180,E1 -5421.002,E2 -5421.002} C_VEL
LIN {X 0,Y 509.869,Z 427.594,A -85,B 0,C 180,E1 -5424.426,E2 -5424.426} C_VEL
LIN {X 0,Y 509.885,Z 427.593,A -85,B 0,C 180,E1 -5427.055,E2 -5427.055} C_VEL
LIN {X 0,Y 509.856,Z 427.603,A -85,B 0,C 180,E1 -5429.751,E2 -5429.751} C_VEL
LIN {X 0,Y 509.874,Z 427.593,A -85,B 0,C 180,E1 -5432.774,E2 -5432.774} C_VEL
LIN {X 0,Y 509.842,Z 427.604,A -85,B 0,C 180,E1 -5435.581,E2 -5435.581} C_VEL
LIN {X 0,Y 509.85,Z 427.598,A -85,B 0,C 180,E1 -5438.338,E2 -5438.338} C_VEL
LIN {X 0,Y 509.856,Z 427.6,A -85,B 0,C 180,E1 -5441.425,E2 -5441.425} C_VEL
LIN {X 0,Y 509.856,Z 427.596,A -85,B 0,C 180,E1 -5444.668,E2 -5444.668} C_VEL
LIN {X 0,Y 509.86,Z 427.6,A -85,B 0,C 180,E1 -5448.103,E2 -5448.103} C_VEL
LIN {X 0,Y 509.846,Z 427.598,A -85,B 0,C 180,E1 -5450.648,E2 -5450.648} C_VEL
LIN {X 0,Y 509.825,Z 427.604,A -85,B 0,C 180,E1 -5453.647,E2 -5453.647} C_VEL
LIN {X 0,Y 509.859,Z 427.599,A -85,B 0,C 180,E1 -5456.539,E2 -5456.539} C_VEL
LIN {X 0,Y 509.846,Z 427.604,A -85,B 0,C 180,E1 -5459.334,E2 -5459.334} C_VEL
LIN {X 0,Y 509.897,Z 427.719,A -85,B 0,C 180,E1 -5461.393,E2 -5461.393} C_VEL
LIN {X 0,Y 513.207,Z 441.896,A -85,B 0,C 180,E1 -5463.572,E2 -5463.572} C_VEL
LIN {X 0,Y 512.638,Z 459.213,A -85,B 0,C 180,E1 -5465.93,E2 -5465.93} C_VEL
LIN {X 0,Y 512.111,Z 473.887,A -85,B 0,C 180,E1 -5467.899,E2 -5467.899} C_VEL
LIN {X 0,Y 515.305,Z 490.877,A -85,B 0,C 180,E1 -5468.298,E2 -5468.298} C_VEL
LIN {X 0,Y 514.155,Z 639.785,A -85,B 0,C 180,E1 -5470.447,E2 -5470.447} C_VEL
LIN {X 0,Y 513.801,Z 655.703,A -85,B 0,C 180,E1 -5470.835,E2 -5470.835} C_VEL
LIN {X 0,Y 513.347,Z 671.144,A -85,B 0,C 180,E1 -5471.388,E2 -5471.388} C_VEL
LIN {X 0,Y 512.839,Z 684.962,A -85,B 0,C 180,E1 -5472.04,E2 -5472.04} C_VEL
LIN {X 0,Y 512.293,Z 698.512,A -85,B 0,C 180,E1 -5472.845,E2 -5472.845} C_VEL
LIN {X 0,Y 511.732,Z 712.301,A -85,B 0,C 180,E1 -5473.852,E2 -5473.852} C_VEL
LIN {X 0,Y 511.11,Z 724.777,A -85,B 0,C 180,E1 -5474.957,E2 -5474.957} C_VEL
LIN {X 0,Y 510.59,Z 737.015,A -85,B 0,C 180,E1 -5476.264,E2 -5476.264} C_VEL
LIN {X 0,Y 510.146,Z 747.894,A -85,B 0,C 180,E1 -5477.67,E2 -5477.67} C_VEL
LIN {X 0,Y 509.878,Z 756.955,A -85,B 0,C 180,E1 -5479.075,E2 -5479.075} C_VEL
LIN {X 0,Y 509.548,Z 764.465,A -85,B 0,C 180,E1 -5480.473,E2 -5480.473} C_VEL
LIN {X 0,Y 509.385,Z 771.477,A -85,B 0,C 180,E1 -5482.069,E2 -5482.069} C_VEL
LIN {X 0,Y 509.257,Z 776.989,A -85,B 0,C 180,E1 -5483.661,E2 -5483.661} C_VEL
LIN {X 0,Y 509.159,Z 781.155,A -85,B 0,C 180,E1 -5485.249,E2 -5485.249} C_VEL
LIN {X 0,Y 509.188,Z 784.078,A -85,B 0,C 180,E1 -5486.835,E2 -5486.835} C_VEL
LIN {X 0,Y 509.109,Z 785.818,A -85,B 0,C 180,E1 -5488.418,E2 -5488.418} C_VEL
LIN {X 0,Y 509.062,Z 786.414,A -85,B 0,C 180,E1 -5490,E2 -5490} C_VEL
LIN {X 0,Y 509.109,Z 785.816,A -85,B 0,C 180,E1 -5491.582,E2 -5491.582} C_VEL
LIN {X 0,Y 509.188,Z 784.073,A -85,B 0,C 180,E1 -5493.164,E2 -5493.164} C_VEL
LIN {X 0,Y 509.158,Z 781.152,A -85,B 0,C 180,E1 -5494.75,E2 -5494.75} C_VEL
LIN {X 0,Y 509.256,Z 776.991,A -85,B 0,C 180,E1 -5496.338,E2 -5496.338} C_VEL
LIN {X 0,Y 509.384,Z 771.474,A -85,B 0,C 180,E1 -5497.93,E2 -5497.93} C_VEL
LIN {X 0,Y 509.547,Z 764.451,A -85,B 0,C 180,E1 -5499.526,E2 -5499.526} C_VEL
LIN {X 0,Y 509.884,Z 755.715,A -85,B 0,C 180,E1 -5501.126,E2 -5501.126} C_VEL
LIN {X 0,Y 510.195,Z 746.43,A -85,B 0,C 180,E1 -5502.53,E2 -5502.53} C_VEL
LIN {X 0,Y 510.589,Z 736.991,A -85,B 0,C 180,E1 -5503.735,E2 -5503.735} C_VEL
LIN {X 0,Y 511.113,Z 724.752,A -85,B 0,C 180,E1 -5505.042,E2 -5505.042} C_VEL
LIN {X 0,Y 511.726,Z 712.274,A -85,B 0,C 180,E1 -5506.147,E2 -5506.147} C_VEL
LIN {X 0,Y 512.208,Z 699.996,A -85,B 0,C 180,E1 -5507.054,E2 -5507.054} C_VEL
LIN {X 0,Y 512.746,Z 686.735,A -85,B 0,C 180,E1 -5507.859,E2 -5507.859} C_VEL
LIN {X 0,Y 513.317,Z 672.235,A -85,B 0,C 180,E1 -5508.561,E2 -5508.561} C_VEL
LIN {X 0,Y 513.722,Z 657.269,A -85,B 0,C 180,E1 -5509.113,E2 -5509.113} C_VEL
LIN {X 0,Y 514.068,Z 643.164,A -85,B 0,C 180,E1 -5509.48,E2 -5509.48} C_VEL
LIN {X 0,Y 514.327,Z 620.415,A -85,B 0,C 180,E1 -5509.846,E2 -5509.846} C_VEL
LIN {X 0,Y 515.276,Z 489.952,A -85,B 0,C 180,E1 -5511.715,E2 -5511.715} C_VEL
LIN {X 0,Y 512.083,Z 473.75,A -85,B 0,C 180,E1 -5512.101,E2 -5512.101} C_VEL
LIN {X 0,Y 512.9,Z 451.153,A -85,B 0,C 180,E1 -5515.136,E2 -5515.136} C_VEL
LIN {X 0,Y 513.156,Z 441.706,A -85,B 0,C 180,E1 -5516.429,E2 -5516.429} C_VEL
LIN {X 0,Y 509.895,Z 427.603,A -85,B 0,C 180,E1 -5518.605,E2 -5518.605} C_VEL
LIN {X 0,Y 509.823,Z 427.604,A -85,B 0,C 180,E1 -5521.589,E2 -5521.589} C_VEL
LIN {X 0,Y 509.848,Z 427.604,A -85,B 0,C 180,E1 -5524.413,E2 -5524.413} C_VEL
LIN {X 0,Y 509.816,Z 427.601,A -85,B 0,C 180,E1 -5527.34,E2 -5527.34} C_VEL
LIN {X 0,Y 509.857,Z 427.601,A -85,B 0,C 180,E1 -5530.379,E2 -5530.379} C_VEL
LIN {X 0,Y 509.835,Z 427.597,A -85,B 0,C 180,E1 -5533.064,E2 -5533.064} C_VEL
LIN {X 0,Y 509.824,Z 427.603,A -85,B 0,C 180,E1 -5535.792,E2 -5535.792} C_VEL
LIN {X 0,Y 509.853,Z 427.602,A -85,B 0,C 180,E1 -5538.574,E2 -5538.574} C_VEL
LIN {X 0,Y 509.845,Z 427.6,A -85,B 0,C 180,E1 -5541.786,E2 -5541.786} C_VEL
LIN {X 0,Y 509.841,Z 427.602,A -85,B 0,C 180,E1 -5544.623,E2 -5544.623} C_VEL
LIN {X 0,Y 509.86,Z 427.594,A -85,B 0,C 180,E1 -5547.481,E2 -5547.481} C_VEL
LIN {X 0,Y 509.851,Z 427.602,A -85,B 0,C 180,E1 -5550.273,E2 -5550.273} C_VEL
LIN {X 0,Y 509.88,Z 427.592,A -85,B 0,C 180,E1 -5552.944,E2 -5552.944} C_VEL
LIN {X 0,Y 509.863,Z 427.595,A -85,B 0,C 180,E1 -5555.574,E2 -5555.574} C_VEL
LIN {X 0,Y 509.816,Z 427.607,A -85,B 0,C 180,E1 -5558.149,E2 -5558.149} C_VEL
LIN {X 0,Y 509.858,Z 427.6,A -85,B 0,C 180,E1 -5560.682,E2 -5560.682} C_VEL
LIN {X 0,Y 509.879,Z 427.59,A -85,B 0,C 180,E1 -5563.175,E2 -5563.175} C_VEL
LIN {X 0,Y 509.857,Z 427.596,A -85,B 0,C 180,E1 -5565.634,E2 -5565.634} C_VEL
LIN {X 0,Y 509.915,Z 427.59,A -85,B 0,C 180,E1 -5568.875,E2 -5568.875} C_VEL
LIN {X 0,Y 509.944,Z 427.589,A -85,B 0,C 180,E1 -5572.079,E2 -5572.079} C_VEL
LIN {X 0,Y 509.976,Z 427.586,A -85,B 0,C 180,E1 -5574.464,E2 -5574.464} C_VEL
LIN {X 0,Y 510.049,Z 427.57,A -85,B 0,C 180,E1 -5577.631,E2 -5577.631} C_VEL
LIN {X 0,Y 510.058,Z 427.571,A -85,B 0,C 180,E1 -5580.79,E2 -5580.79} C_VEL
LIN {X 0,Y 509.952,Z 427.584,A -85,B 0,C 180,E1 -5583.16,E2 -5583.16} C_VEL
LIN {X 0,Y 509.975,Z 427.588,A -85,B 0,C 180,E1 -5586.33,E2 -5586.33} C_VEL
LIN {X 0,Y 509.911,Z 427.593,A -85,B 0,C 180,E1 -5588.72,E2 -5588.72} C_VEL
LIN {X 0,Y 509.897,Z 427.592,A -85,B 0,C 180,E1 -5591.932,E2 -5591.932} C_VEL
LIN {X 0,Y 509.886,Z 427.592,A -85,B 0,C 180,E1 -5595.242,E2 -5595.242} C_VEL
LIN {X 0,Y 509.882,Z 427.596,A -85,B 0,C 180,E1 -5598.002,E2 -5598.002} C_VEL
LIN {X 0,Y 509.845,Z 427.598,A -85,B 0,C 180,E1 -5601.002,E2 -5601.002} C_VEL
LIN {X 0,Y 509.831,Z 427.6,A -85,B 0,C 180,E1 -5603.564,E2 -5603.564} C_VEL
LIN {X 0,Y 509.908,Z 427.594,A -85,B 0,C 180,E1 -5606.38,E2 -5606.38} C_VEL
LIN {X 0,Y 509.881,Z 427.596,A -85,B 0,C 180,E1 -5608.844,E2 -5608.844} C_VEL
LIN {X 0,Y 509.822,Z 427.601,A -85,B 0,C 180,E1 -5611.59,E2 -5611.59} C_VEL
LIN {X 0,Y 509.85,Z 427.603,A -85,B 0,C 180,E1 -5614.414,E2 -5614.414} C_VEL
LIN {X 0,Y 509.816,Z 427.604,A -85,B 0,C 180,E1 -5617.341,E2 -5617.341} C_VEL
LIN {X 0,Y 509.858,Z 427.602,A -85,B 0,C 180,E1 -5620.381,E2 -5620.381} C_VEL
LIN {X 0,Y 509.881,Z 427.651,A -85,B 0,C 180,E1 -5622.714,E2 -5622.714} C_VEL
LIN {X 0,Y 512.284,Z 438.988,A -85,B 0,C 180,E1 -5624.676,E2 -5624.676} C_VEL
LIN {X 0,Y 512.016,Z 447.086,A -85,B 0,C 180,E1 -5625.95,E2 -5625.95} C_VEL
LIN {X 0,Y 515.409,Z 462.909,A -85,B 0,C 180,E1 -5626.348,E2 -5626.348} C_VEL
LIN {X 0,Y 515.068,Z 498.627,A -85,B 0,C 180,E1 -5626.861,E2 -5626.861} C_VEL
LIN {X 0,Y 514.297,Z 504.478,A -85,B 0,C 180,E1 -5626.913,E2 -5626.913} C_VEL
LIN {X 0,Y 508.88,Z 523.549,A -85,B 0,C 180,E1 -5626.959,E2 -5626.959} C_VEL
LIN {X 0,Y 508.246,Z 529.394,A -85,B 0,C 180,E1 -5627.018,E2 -5627.018} C_VEL
LIN {X 0,Y 507.526,Z 612.424,A -85,B 0,C 180,E1 -5628.244,E2 -5628.244} C_VEL
LIN {X 0,Y 507.182,Z 627.572,A -85,B 0,C 180,E1 -5628.623,E2 -5628.623} C_VEL
LIN {X 0,Y 506.751,Z 641.504,A -85,B 0,C 180,E1 -5629.125,E2 -5629.125} C_VEL
LIN {X 0,Y 506.229,Z 655.413,A -85,B 0,C 180,E1 -5629.78,E2 -5629.78} C_VEL
LIN {X 0,Y 505.708,Z 667.987,A -85,B 0,C 180,E1 -5630.522,E2 -5630.522} C_VEL
LIN {X 0,Y 505.064,Z 681.406,A -85,B 0,C 180,E1 -5631.488,E2 -5631.488} C_VEL
LIN {X 0,Y 504.486,Z 693.739,A -85,B 0,C 180,E1 -5632.568,E2 -5632.568} C_VEL
LIN {X 0,Y 503.962,Z 704.019,A -85,B 0,C 180,E1 -5633.634,E2 -5633.634} C_VEL
LIN {X 0,Y 503.484,Z 713.952,A -85,B 0,C 180,E1 -5634.846,E2 -5634.846} C_VEL
LIN {X 0,Y 503.011,Z 723.702,A -85,B 0,C 180,E1 -5636.264,E2 -5636.264} C_VEL
LIN {X 0,Y 502.706,Z 731.791,A -85,B 0,C 180,E1 -5637.677,E2 -5637.677} C_VEL
LIN {X 0,Y 502.417,Z 739.413,A -85,B 0,C 180,E1 -5639.299,E2 -5639.299} C_VEL
LIN {X 0,Y 502.252,Z 744.626,A -85,B 0,C 180,E1 -5640.676,E2 -5640.676} C_VEL
LIN {X 0,Y 502.176,Z 748.322,A -85,B 0,C 180,E1 -5641.848,E2 -5641.848} C_VEL
LIN {X 0,Y 502.035,Z 752.578,A -85,B 0,C 180,E1 -5643.63,E2 -5643.63} C_VEL
LIN {X 0,Y 501.998,Z 755.446,A -85,B 0,C 180,E1 -5645.506,E2 -5645.506} C_VEL
LIN {X 0,Y 501.972,Z 756.782,A -85,B 0,C 180,E1 -5647.526,E2 -5647.526} C_VEL
LIN {X 0,Y 501.95,Z 756.765,A -85,B 0,C 180,E1 -5648.652,E2 -5648.652} C_VEL
LIN {X 0,Y 502.007,Z 755.659,A -85,B 0,C 180,E1 -5650.368,E2 -5650.368} C_VEL
LIN {X 0,Y 502.053,Z 753.114,A -85,B 0,C 180,E1 -5652.158,E2 -5652.158} C_VEL
LIN {X 0,Y 502.146,Z 749.613,A -85,B 0,C 180,E1 -5653.745,E2 -5653.745} C_VEL
LIN {X 0,Y 502.283,Z 744.606,A -85,B 0,C 180,E1 -5655.413,E2 -5655.413} C_VEL
LIN {X 0,Y 502.446,Z 738.172,A -85,B 0,C 180,E1 -5657.068,E2 -5657.068} C_VEL
LIN {X 0,Y 502.783,Z 730.116,A -85,B 0,C 180,E1 -5658.715,E2 -5658.715} C_VEL
LIN {X 0,Y 503.111,Z 721.58,A -85,B 0,C 180,E1 -5660.148,E2 -5660.148} C_VEL
LIN {X 0,Y 503.576,Z 711.348,A -85,B 0,C 180,E1 -5661.574,E2 -5661.574} C_VEL
LIN {X 0,Y 504.117,Z 700.902,A -85,B 0,C 180,E1 -5662.793,E2 -5662.793} C_VEL
LIN {X 0,Y 504.66,Z 689.607,A -85,B 0,C 180,E1 -5663.905,E2 -5663.905} C_VEL
LIN {X 0,Y 505.254,Z 677.383,A -85,B 0,C 180,E1 -5664.913,E2 -5664.913} C_VEL
LIN {X 0,Y 505.897,Z 664.034,A -85,B 0,C 180,E1 -5665.818,E2 -5665.818} C_VEL
LIN {X 0,Y 506.459,Z 650.271,A -85,B 0,C 180,E1 -5666.57,E2 -5666.57} C_VEL
LIN {X 0,Y 506.95,Z 635.292,A -85,B 0,C 180,E1 -5667.205,E2 -5667.205} C_VEL
LIN {X 0,Y 507.348,Z 619.302,A -85,B 0,C 180,E1 -5667.693,E2 -5667.693} C_VEL
LIN {X 0,Y 507.578,Z 603.946,A -85,B 0,C 180,E1 -5667.992,E2 -5667.992} C_VEL
LIN {X 0,Y 508.753,Z 462.939,A -85,B 0,C 180,E1 -5670.041,E2 -5670.041} C_VEL
LIN {X 0,Y 505.197,Z 447.14,A -85,B 0,C 180,E1 -5670.456,E2 -5670.456} C_VEL
LIN {X 0,Y 505.324,Z 440.006,A -85,B 0,C 180,E1 -5671.594,E2 -5671.594} C_VEL
LIN {X 0,Y 503.437,Z 430.764,A -85,B 0,C 180,E1 -5673.201,E2 -5673.201} C_VEL
LIN {X 0,Y 502.864,Z 428.474,A -85,B 0,C 180,E1 -5673.631,E2 -5673.631} C_VEL
LIN {X 0,Y 502.891,Z 428.467,A -85,B 0,C 180,E1 -5676.42,E2 -5676.42} C_VEL
LIN {X 0,Y 502.878,Z 428.468,A -85,B 0,C 180,E1 -5678.844,E2 -5678.844} C_VEL
LIN {X 0,Y 502.898,Z 428.467,A -85,B 0,C 180,E1 -5682.101,E2 -5682.101} C_VEL
LIN {X 0,Y 502.853,Z 428.475,A -85,B 0,C 180,E1 -5685.4,E2 -5685.4} C_VEL
LIN {X 0,Y 502.845,Z 428.472,A -85,B 0,C 180,E1 -5688.12,E2 -5688.12} C_VEL
LIN {X 0,Y 502.833,Z 428.47,A -85,B 0,C 180,E1 -5690.536,E2 -5690.536} C_VEL
LIN {X 0,Y 502.802,Z 428.477,A -85,B 0,C 180,E1 -5693.04,E2 -5693.04} C_VEL
LIN {X 0,Y 502.845,Z 428.477,A -85,B 0,C 180,E1 -5695.675,E2 -5695.675} C_VEL
LIN {X 0,Y 502.844,Z 428.467,A -85,B 0,C 180,E1 -5698.373,E2 -5698.373} C_VEL
LIN {X 0,Y 502.801,Z 428.482,A -85,B 0,C 180,E1 -5701.499,E2 -5701.499} C_VEL
LIN {X 0,Y 502.808,Z 428.474,A -85,B 0,C 180,E1 -5704.444,E2 -5704.444} C_VEL
LIN {X 0,Y 502.784,Z 428.478,A -85,B 0,C 180,E1 -5707.178,E2 -5707.178} C_VEL
LIN {X 0,Y 502.791,Z 428.479,A -85,B 0,C 180,E1 -5710.015,E2 -5710.015} C_VEL
LIN {X 0,Y 502.806,Z 428.473,A -85,B 0,C 180,E1 -5712.199,E2 -5712.199} C_VEL
LIN {X 0,Y 502.803,Z 428.479,A -85,B 0,C 180,E1 -5715.468,E2 -5715.468} C_VEL
LIN {X 0,Y 502.829,Z 428.467,A -85,B 0,C 180,E1 -5719.004,E2 -5719.004} C_VEL
LIN {X 0,Y 502.797,Z 428.477,A -85,B 0,C 180,E1 -5722.046,E2 -5722.046} C_VEL
LIN {X 0,Y 502.812,Z 428.47,A -85,B 0,C 180,E1 -5725.035,E2 -5725.035} C_VEL
LIN {X 0,Y 502.786,Z 428.48,A -85,B 0,C 180,E1 -5727.915,E2 -5727.915} C_VEL
LIN {X 0,Y 502.825,Z 428.466,A -85,B 0,C 180,E1 -5730.712,E2 -5730.712} C_VEL
LIN {X 0,Y 502.882,Z 428.469,A -85,B 0,C 180,E1 -5733.435,E2 -5733.435} C_VEL
LIN {X 0,Y 502.786,Z 428.472,A -85,B 0,C 180,E1 -5736.086,E2 -5736.086} C_VEL
LIN {X 0,Y 502.784,Z 428.475,A -85,B 0,C 180,E1 -5738.689,E2 -5738.689} C_VEL
LIN {X 0,Y 502.83,Z 428.473,A -85,B 0,C 180,E1 -5741.248,E2 -5741.248} C_VEL
LIN {X 0,Y 502.823,Z 428.473,A -85,B 0,C 180,E1 -5743.767,E2 -5743.767} C_VEL
LIN {X 0,Y 502.831,Z 428.472,A -85,B 0,C 180,E1 -5746.254,E2 -5746.254} C_VEL
LIN {X 0,Y 502.877,Z 428.462,A -85,B 0,C 180,E1 -5748.717,E2 -5748.717} C_VEL
LIN {X 0,Y 502.902,Z 428.466,A -85,B 0,C 180,E1 -5751.966,E2 -5751.966} C_VEL
LIN {X 0,Y 502.938,Z 428.457,A -85,B 0,C 180,E1 -5754.386,E2 -5754.386} C_VEL
LIN {X 0,Y 503.024,Z 428.447,A -85,B 0,C 180,E1 -5757.598,E2 -5757.598} C_VEL
LIN {X 0,Y 503.027,Z 428.451,A -85,B 0,C 180,E1 -5760,E2 -5760} C_VEL
LIN {X 0,Y 503.024,Z 428.444,A -85,B 0,C 180,E1 -5762.402,E2 -5762.402} C_VEL
LIN {X 0,Y 502.937,Z 428.456,A -85,B 0,C 180,E1 -5765.613,E2 -5765.613} C_VEL
LIN {X 0,Y 502.901,Z 428.466,A -85,B 0,C 180,E1 -5768.033,E2 -5768.033} C_VEL
LIN {X 0,Y 502.876,Z 428.464,A -85,B 0,C 180,E1 -5771.283,E2 -5771.283} C_VEL
LIN {X 0,Y 502.844,Z 428.469,A -85,B 0,C 180,E1 -5774.571,E2 -5774.571} C_VEL
LIN {X 0,Y 502.861,Z 428.466,A -85,B 0,C 180,E1 -5777.907,E2 -5777.907} C_VEL
LIN {X 0,Y 502.828,Z 428.471,A -85,B 0,C 180,E1 -5780.536,E2 -5780.536} C_VEL
LIN {X 0,Y 502.794,Z 428.475,A -85,B 0,C 180,E1 -5783.04,E2 -5783.04} C_VEL
LIN {X 0,Y 502.84,Z 428.477,A -85,B 0,C 180,E1 -5785.675,E2 -5785.675} C_VEL
LIN {X 0,Y 502.84,Z 428.47,A -85,B 0,C 180,E1 -5788.373,E2 -5788.373} C_VEL
LIN {X 0,Y 502.793,Z 428.48,A -85,B 0,C 180,E1 -5791.499,E2 -5791.499} C_VEL
LIN {X 0,Y 502.806,Z 428.474,A -85,B 0,C 180,E1 -5794.445,E2 -5794.445} C_VEL
LIN {X 0,Y 502.781,Z 428.479,A -85,B 0,C 180,E1 -5797.178,E2 -5797.178} C_VEL
LIN {X 0,Y 502.788,Z 428.481,A -85,B 0,C 180,E1 -5800.015,E2 -5800.015} C_VEL
LIN {X 0,Y 502.802,Z 428.477,A -85,B 0,C 180,E1 -5802.199,E2 -5802.199} C_VEL
LIN {X 0,Y 502.801,Z 428.48,A -85,B 0,C 180,E1 -5805.468,E2 -5805.468} C_VEL
LIN {X 0,Y 502.83,Z 428.478,A -85,B 0,C 180,E1 -5807.864,E2 -5807.864} C_VEL
LIN {X 0,Y 502.802,Z 428.476,A -85,B 0,C 180,E1 -5811.024,E2 -5811.024} C_VEL
LIN {X 0,Y 502.775,Z 428.484,A -85,B 0,C 180,E1 -5814.169,E2 -5814.169} C_VEL
LIN {X 0,Y 502.833,Z 428.475,A -85,B 0,C 180,E1 -5816.993,E2 -5816.993} C_VEL
LIN {X 0,Y 502.815,Z 428.481,A -85,B 0,C 180,E1 -5820.065,E2 -5820.065} C_VEL
LIN {X 0,Y 502.859,Z 428.641,A -85,B 0,C 180,E1 -5821.116,E2 -5821.116} C_VEL
LIN {X 0,Y 506.35,Z 443.51,A -85,B 0,C 180,E1 -5823.441,E2 -5823.441} C_VEL
LIN {X 0,Y 506.035,Z 454.29,A -85,B 0,C 180,E1 -5824.938,E2 -5824.938} C_VEL
LIN {X 0,Y 505.27,Z 473.656,A -85,B 0,C 180,E1 -5827.58,E2 -5827.58} C_VEL
LIN {X 0,Y 508.643,Z 490.68,A -85,B 0,C 180,E1 -5827.999,E2 -5827.999} C_VEL
LIN {X 0,Y 507.577,Z 626.045,A -85,B 0,C 180,E1 -5829.965,E2 -5829.965} C_VEL
LIN {X 0,Y 507.356,Z 644.276,A -85,B 0,C 180,E1 -5830.281,E2 -5830.281} C_VEL
LIN {X 0,Y 506.977,Z 659.207,A -85,B 0,C 180,E1 -5830.696,E2 -5830.696} C_VEL
LIN {X 0,Y 506.523,Z 673.347,A -85,B 0,C 180,E1 -5831.241,E2 -5831.241} C_VEL
LIN {X 0,Y 505.975,Z 686.559,A -85,B 0,C 180,E1 -5831.893,E2 -5831.893} C_VEL
LIN {X 0,Y 505.388,Z 699.814,A -85,B 0,C 180,E1 -5832.708,E2 -5832.708} C_VEL
LIN {X 0,Y 504.798,Z 713.304,A -85,B 0,C 180,E1 -5833.728,E2 -5833.728} C_VEL
LIN {X 0,Y 504.132,Z 725.583,A -85,B 0,C 180,E1 -5834.847,E2 -5834.847} C_VEL
LIN {X 0,Y 503.634,Z 736.797,A -85,B 0,C 180,E1 -5836.071,E2 -5836.071} C_VEL
LIN {X 0,Y 503.141,Z 747.678,A -85,B 0,C 180,E1 -5837.496,E2 -5837.496} C_VEL
LIN {X 0,Y 502.841,Z 756.741,A -85,B 0,C 180,E1 -5838.92,E2 -5838.92} C_VEL
LIN {X 0,Y 502.472,Z 764.253,A -85,B 0,C 180,E1 -5840.337,E2 -5840.337} C_VEL
LIN {X 0,Y 502.3,Z 771.267,A -85,B 0,C 180,E1 -5841.957,E2 -5841.957} C_VEL
LIN {X 0,Y 502.185,Z 776.781,A -85,B 0,C 180,E1 -5843.571,E2 -5843.571} C_VEL
LIN {X 0,Y 502.081,Z 780.948,A -85,B 0,C 180,E1 -5845.182,E2 -5845.182} C_VEL
LIN {X 0,Y 502.107,Z 783.871,A -85,B 0,C 180,E1 -5846.79,E2 -5846.79} C_VEL
LIN {X 0,Y 502.033,Z 785.612,A -85,B 0,C 180,E1 -5848.395,E2 -5848.395} C_VEL
LIN {X 0,Y 501.977,Z 786.207,A -85,B 0,C 180,E1 -5850,E2 -5850} C_VEL
LIN {X 0,Y 502.032,Z 785.608,A -85,B 0,C 180,E1 -5851.604,E2 -5851.604} C_VEL
LIN {X 0,Y 502.107,Z 783.863,A -85,B 0,C 180,E1 -5853.209,E2 -5853.209} C_VEL
LIN {X 0,Y 502.081,Z 780.94,A -85,B 0,C 180,E1 -5854.817,E2 -5854.817} C_VEL
LIN {X 0,Y 502.184,Z 776.65,A -85,B 0,C 180,E1 -5856.468,E2 -5856.468} C_VEL
LIN {X 0,Y 502.299,Z 771.256,A -85,B 0,C 180,E1 -5858.042,E2 -5858.042} C_VEL
LIN {X 0,Y 502.471,Z 764.23,A -85,B 0,C 180,E1 -5859.662,E2 -5859.662} C_VEL
LIN {X 0,Y 502.831,Z 756.715,A -85,B 0,C 180,E1 -5861.08,E2 -5861.08} C_VEL
LIN {X 0,Y 503.144,Z 747.65,A -85,B 0,C 180,E1 -5862.503,E2 -5862.503} C_VEL
LIN {X 0,Y 503.608,Z 736.758,A -85,B 0,C 180,E1 -5863.929,E2 -5863.929} C_VEL
LIN {X 0,Y 504.188,Z 724.514,A -85,B 0,C 180,E1 -5865.254,E2 -5865.254} C_VEL
LIN {X 0,Y 504.834,Z 712.029,A -85,B 0,C 180,E1 -5866.373,E2 -5866.373} C_VEL
LIN {X 0,Y 505.37,Z 699.748,A -85,B 0,C 180,E1 -5867.292,E2 -5867.292} C_VEL
LIN {X 0,Y 505.936,Z 686.479,A -85,B 0,C 180,E1 -5868.108,E2 -5868.108} C_VEL
LIN {X 0,Y 506.544,Z 672.168,A -85,B 0,C 180,E1 -5868.809,E2 -5868.809} C_VEL
LIN {X 0,Y 506.99,Z 657.066,A -85,B 0,C 180,E1 -5869.374,E2 -5869.374} C_VEL
LIN {X 0,Y 507.367,Z 642.853,A -85,B 0,C 180,E1 -5869.748,E2 -5869.748} C_VEL
LIN {X 0,Y 507.65,Z 620.056,A -85,B 0,C 180,E1 -5870.118,E2 -5870.118} C_VEL
LIN {X 0,Y 508.675,Z 490.946,A -85,B 0,C 180,E1 -5871.993,E2 -5871.993} C_VEL
LIN {X 0,Y 505.22,Z 473.521,A -85,B 0,C 180,E1 -5872.417,E2 -5872.417} C_VEL
LIN {X 0,Y 506.144,Z 450.871,A -85,B 0,C 180,E1 -5875.505,E2 -5875.505} C_VEL
LIN {X 0,Y 506.311,Z 443.318,A -85,B 0,C 180,E1 -5876.559,E2 -5876.559} C_VEL
LIN {X 0,Y 502.858,Z 428.477,A -85,B 0,C 180,E1 -5878.883,E2 -5878.883} C_VEL
LIN {X 0,Y 502.785,Z 428.483,A -85,B 0,C 180,E1 -5882.084,E2 -5882.084} C_VEL
LIN {X 0,Y 502.804,Z 428.476,A -85,B 0,C 180,E1 -5884.964,E2 -5884.964} C_VEL
LIN {X 0,Y 502.793,Z 428.478,A -85,B 0,C 180,E1 -5887.953,E2 -5887.953} C_VEL
LIN {X 0,Y 502.822,Z 428.474,A -85,B 0,C 180,E1 -5891.065,E2 -5891.065} C_VEL
LIN {X 0,Y 502.777,Z 428.476,A -85,B 0,C 180,E1 -5893.375,E2 -5893.375} C_VEL
LIN {X 0,Y 502.784,Z 428.48,A -85,B 0,C 180,E1 -5895.661,E2 -5895.661} C_VEL
LIN {X 0,Y 502.813,Z 428.475,A -85,B 0,C 180,E1 -5899.004,E2 -5899.004} C_VEL
LIN {X 0,Y 502.788,Z 428.482,A -85,B 0,C 180,E1 -5902.046,E2 -5902.046} C_VEL
LIN {X 0,Y 502.804,Z 428.475,A -85,B 0,C 180,E1 -5905.035,E2 -5905.035} C_VEL
LIN {X 0,Y 502.781,Z 428.479,A -85,B 0,C 180,E1 -5907.915,E2 -5907.915} C_VEL
LIN {X 0,Y 502.817,Z 428.476,A -85,B 0,C 180,E1 -5910.712,E2 -5910.712} C_VEL
LIN {X 0,Y 502.874,Z 428.464,A -85,B 0,C 180,E1 -5913.435,E2 -5913.435} C_VEL
LIN {X 0,Y 502.785,Z 428.481,A -85,B 0,C 180,E1 -5916.086,E2 -5916.086} C_VEL
LIN {X 0,Y 502.777,Z 428.479,A -85,B 0,C 180,E1 -5918.689,E2 -5918.689} C_VEL
LIN {X 0,Y 502.823,Z 428.472,A -85,B 0,C 180,E1 -5921.248,E2 -5921.248} C_VEL
LIN {X 0,Y 502.816,Z 428.471,A -85,B 0,C 180,E1 -5923.767,E2 -5923.767} C_VEL
LIN {X 0,Y 502.824,Z 428.478,A -85,B 0,C 180,E1 -5926.255,E2 -5926.255} C_VEL
LIN {X 0,Y 502.885,Z 428.467,A -85,B 0,C 180,E1 -5928.717,E2 -5928.717} C_VEL
LIN {X 0,Y 502.895,Z 428.465,A -85,B 0,C 180,E1 -5931.967,E2 -5931.967} C_VEL
LIN {X 0,Y 502.932,Z 428.463,A -85,B 0,C 180,E1 -5934.387,E2 -5934.387} C_VEL
LIN {X 0,Y 503.019,Z 428.446,A -85,B 0,C 180,E1 -5937.598,E2 -5937.598} C_VEL
LIN {X 0,Y 503.019,Z 428.451,A -85,B 0,C 180,E1 -5940,E2 -5940} C_VEL
LIN {X 0,Y 503.019,Z 428.454,A -85,B 0,C 180,E1 -5942.402,E2 -5942.402} C_VEL
LIN {X 0,Y 502.935,Z 428.457,A -85,B 0,C 180,E1 -5945.614,E2 -5945.614} C_VEL
LIN {X 0,Y 502.895,Z 428.466,A -85,B 0,C 180,E1 -5948.034,E2 -5948.034} C_VEL
LIN {X 0,Y 502.87,Z 428.464,A -85,B 0,C 180,E1 -5951.284,E2 -5951.284} C_VEL
LIN {X 0,Y 502.845,Z 428.476,A -85,B 0,C 180,E1 -5954.571,E2 -5954.571} C_VEL
LIN {X 0,Y 502.856,Z 428.47,A -85,B 0,C 180,E1 -5957.907,E2 -5957.907} C_VEL
LIN {X 0,Y 502.822,Z 428.479,A -85,B 0,C 180,E1 -5960.537,E2 -5960.537} C_VEL
LIN {X 0,Y 502.791,Z 428.478,A -85,B 0,C 180,E1 -5963.041,E2 -5963.041} C_VEL
LIN {X 0,Y 502.836,Z 428.473,A -85,B 0,C 180,E1 -5965.676,E2 -5965.676} C_VEL
LIN {X 0,Y 502.837,Z 428.48,A -85,B 0,C 180,E1 -5968.373,E2 -5968.373} C_VEL
LIN {X 0,Y 502.792,Z 428.477,A -85,B 0,C 180,E1 -5971.5,E2 -5971.5} C_VEL
LIN {X 0,Y 502.803,Z 428.481,A -85,B 0,C 180,E1 -5974.446,E2 -5974.446} C_VEL
LIN {X 0,Y 502.778,Z 428.482,A -85,B 0,C 180,E1 -5977.179,E2 -5977.179} C_VEL
LIN {X 0,Y 502.823,Z 428.479,A -85,B 0,C 180,E1 -5980.012,E2 -5980.012} C_VEL
LIN {X 0,Y 502.827,Z 428.521,A -85,B 0,C 180,E1 -5982.442,E2 -5982.442} C_VEL
LIN {X 0,Y 505.351,Z 439.93,A -85,B 0,C 180,E1 -5984.45,E2 -5984.45} C_VEL
LIN {X 0,Y 505.199,Z 447.348,A -85,B 0,C 180,E1 -5985.641,E2 -5985.641} C_VEL
LIN {X 0,Y 508.805,Z 463.281,A -85,B 0,C 180,E1 -5986.054,E2 -5986.054} C_VEL
LIN {X 0,Y 508.246,Z 529.394,A -85,B 0,C 180,E1 -5987.018,E2 -5987.018} C_VEL
LIN {X 0,Y 507.574,Z 535.242,A -85,B 0,C 180,E1 -5987.076,E2 -5987.076} C_VEL
LIN {X 0,Y 501.995,Z 554.281,A -85,B 0,C 180,E1 -5987.118,E2 -5987.118} C_VEL
LIN {X 0,Y 501.33,Z 560.128,A -85,B 0,C 180,E1 -5987.177,E2 -5987.177} C_VEL
LIN {X 0,Y 500.837,Z 613.097,A -85,B 0,C 180,E1 -5987.98,E2 -5987.98} C_VEL
LIN {X 0,Y 500.469,Z 628.561,A -85,B 0,C 180,E1 -5988.381,E2 -5988.381} C_VEL
LIN {X 0,Y 500.028,Z 642.427,A -85,B 0,C 180,E1 -5988.892,E2 -5988.892} C_VEL
LIN {X 0,Y 499.438,Z 657.007,A -85,B 0,C 180,E1 -5989.599,E2 -5989.599} C_VEL
LIN {X 0,Y 498.835,Z 669.981,A -85,B 0,C 180,E1 -5990.394,E2 -5990.394} C_VEL
LIN {X 0,Y 498.157,Z 683.066,A -85,B 0,C 180,E1 -5991.372,E2 -5991.372} C_VEL
LIN {X 0,Y 497.557,Z 695.227,A -85,B 0,C 180,E1 -5992.475,E2 -5992.475} C_VEL
LIN {X 0,Y 496.883,Z 706.794,A -85,B 0,C 180,E1 -5993.729,E2 -5993.729} C_VEL
LIN {X 0,Y 496.401,Z 717.317,A -85,B 0,C 180,E1 -5995.1,E2 -5995.1} C_VEL
LIN {X 0,Y 495.903,Z 725.997,A -85,B 0,C 180,E1 -5996.448,E2 -5996.448} C_VEL
LIN {X 0,Y 495.584,Z 733.702,A -85,B 0,C 180,E1 -5997.874,E2 -5997.874} C_VEL
LIN {X 0,Y 495.356,Z 740.07,A -85,B 0,C 180,E1 -5999.286,E2 -5999.286} C_VEL
LIN {X 0,Y 495.183,Z 745.222,A -85,B 0,C 180,E1 -6000.683,E2 -6000.683} C_VEL
LIN {X 0,Y 495.076,Z 749.327,A -85,B 0,C 180,E1 -6002.066,E2 -6002.066} C_VEL
LIN {X 0,Y 494.956,Z 752.56,A -85,B 0,C 180,E1 -6003.452,E2 -6003.452} C_VEL
LIN {X 0,Y 494.901,Z 755.535,A -85,B 0,C 180,E1 -6005.348,E2 -6005.348} C_VEL
LIN {X 0,Y 494.844,Z 756.588,A -85,B 0,C 180,E1 -6006.568,E2 -6006.568} C_VEL
LIN {X 0,Y 494.852,Z 757.037,A -85,B 0,C 180,E1 -6008.331,E2 -6008.331} C_VEL
LIN {X 0,Y 494.896,Z 756.184,A -85,B 0,C 180,E1 -6010.074,E2 -6010.074} C_VEL
LIN {X 0,Y 494.944,Z 754.06,A -85,B 0,C 180,E1 -6011.797,E2 -6011.797} C_VEL
LIN {X 0,Y 495.055,Z 750.646,A -85,B 0,C 180,E1 -6013.506,E2 -6013.506} C_VEL
LIN {X 0,Y 495.199,Z 745.896,A -85,B 0,C 180,E1 -6015.2,E2 -6015.2} C_VEL
LIN {X 0,Y 495.345,Z 739.748,A -85,B 0,C 180,E1 -6016.88,E2 -6016.88} C_VEL
LIN {X 0,Y 495.676,Z 732.02,A -85,B 0,C 180,E1 -6018.551,E2 -6018.551} C_VEL
LIN {X 0,Y 496.015,Z 723.801,A -85,B 0,C 180,E1 -6020.005,E2 -6020.005} C_VEL
LIN {X 0,Y 496.509,Z 713.962,A -85,B 0,C 180,E1 -6021.453,E2 -6021.453} C_VEL
LIN {X 0,Y 497.067,Z 703.906,A -85,B 0,C 180,E1 -6022.69,E2 -6022.69} C_VEL
LIN {X 0,Y 497.7,Z 692.014,A -85,B 0,C 180,E1 -6023.921,E2 -6023.921} C_VEL
LIN {X 0,Y 498.298,Z 680.181,A -85,B 0,C 180,E1 -6024.943,E2 -6024.943} C_VEL
LIN {X 0,Y 499.006,Z 667.354,A -85,B 0,C 180,E1 -6025.861,E2 -6025.861} C_VEL
LIN {X 0,Y 499.587,Z 653.418,A -85,B 0,C 180,E1 -6026.674,E2 -6026.674} C_VEL
LIN {X 0,Y 500.094,Z 639.573,A -85,B 0,C 180,E1 -6027.309,E2 -6027.309} C_VEL
LIN {X 0,Y 500.568,Z 624.071,A -85,B 0,C 180,E1 -6027.838,E2 -6027.838} C_VEL
LIN {X 0,Y 500.863,Z 608.604,A -85,B 0,C 180,E1 -6028.191,E2 -6028.191} C_VEL
LIN {X 0,Y 502.201,Z 464.246,A -85,B 0,C 180,E1 -6030.327,E2 -6030.327} C_VEL
LIN {X 0,Y 498.386,Z 447.26,A -85,B 0,C 180,E1 -6030.788,E2 -6030.788} C_VEL
LIN {X 0,Y 498.52,Z 442.145,A -85,B 0,C 180,E1 -6031.616,E2 -6031.616} C_VEL
LIN {X 0,Y 496.981,Z 434.004,A -85,B 0,C 180,E1 -6033.04,E2 -6033.04} C_VEL
LIN {X 0,Y 495.762,Z 429.358,A -85,B 0,C 180,E1 -6033.912,E2 -6033.912} C_VEL
LIN {X 0,Y 495.843,Z 429.345,A -85,B 0,C 180,E1 -6036.511,E2 -6036.511} C_VEL
LIN {X 0,Y 495.847,Z 429.345,A -85,B 0,C 180,E1 -6038.97,E2 -6038.97} C_VEL
LIN {X 0,Y 495.857,Z 429.343,A -85,B 0,C 180,E1 -6042.275,E2 -6042.275} C_VEL
LIN {X 0,Y 495.812,Z 429.351,A -85,B 0,C 180,E1 -6045.624,E2 -6045.624} C_VEL
LIN {X 0,Y 495.811,Z 429.347,A -85,B 0,C 180,E1 -6048.247,E2 -6048.247} C_VEL
LIN {X 0,Y 495.778,Z 429.349,A -85,B 0,C 180,E1 -6050.756,E2 -6050.756} C_VEL
LIN {X 0,Y 495.757,Z 429.358,A -85,B 0,C 180,E1 -6053.387,E2 -6053.387} C_VEL
LIN {X 0,Y 495.795,Z 429.35,A -85,B 0,C 180,E1 -6056.068,E2 -6056.068} C_VEL
LIN {X 0,Y 495.776,Z 429.347,A -85,B 0,C 180,E1 -6058.815,E2 -6058.815} C_VEL
LIN {X 0,Y 495.763,Z 429.354,A -85,B 0,C 180,E1 -6061.726,E2 -6061.726} C_VEL
LIN {X 0,Y 495.778,Z 429.35,A -85,B 0,C 180,E1 -6064.695,E2 -6064.695} C_VEL
LIN {X 0,Y 495.735,Z 429.357,A -85,B 0,C 180,E1 -6067.561,E2 -6067.561} C_VEL
LIN {X 0,Y 495.77,Z 429.35,A -85,B 0,C 180,E1 -6070.7,E2 -6070.7} C_VEL
LIN {X 0,Y 495.737,Z 429.358,A -85,B 0,C 180,E1 -6073.695,E2 -6073.695} C_VEL
LIN {X 0,Y 495.731,Z 429.356,A -85,B 0,C 180,E1 -6076.305,E2 -6076.305} C_VEL
LIN {X 0,Y 495.782,Z 429.348,A -85,B 0,C 180,E1 -6079.301,E2 -6079.301} C_VEL
LIN {X 0,Y 495.734,Z 429.353,A -85,B 0,C 180,E1 -6082.438,E2 -6082.438} C_VEL
LIN {X 0,Y 495.787,Z 429.35,A -85,B 0,C 180,E1 -6085.457,E2 -6085.457} C_VEL
LIN {X 0,Y 495.757,Z 429.351,A -85,B 0,C 180,E1 -6088.364,E2 -6088.364} C_VEL
LIN {X 0,Y 495.789,Z 429.349,A -85,B 0,C 180,E1 -6091.506,E2 -6091.506} C_VEL
LIN {X 0,Y 495.801,Z 429.35,A -85,B 0,C 180,E1 -6093.932,E2 -6093.932} C_VEL
LIN {X 0,Y 495.76,Z 429.346,A -85,B 0,C 180,E1 -6097.139,E2 -6097.139} C_VEL
LIN {X 0,Y 495.772,Z 429.352,A -85,B 0,C 180,E1 -6100.109,E2 -6100.109} C_VEL
LIN {X 0,Y 495.787,Z 429.343,A -85,B 0,C 180,E1 -6102.681,E2 -6102.681} C_VEL
LIN {X 0,Y 495.79,Z 429.347,A -85,B 0,C 180,E1 -6105.217,E2 -6105.217} C_VEL
LIN {X 0,Y 495.851,Z 429.337,A -85,B 0,C 180,E1 -6108.555,E2 -6108.555} C_VEL
LIN {X 0,Y 495.873,Z 429.343,A -85,B 0,C 180,E1 -6111.852,E2 -6111.852} C_VEL
LIN {X 0,Y 495.896,Z 429.335,A -85,B 0,C 180,E1 -6114.306,E2 -6114.306} C_VEL
LIN {X 0,Y 495.993,Z 429.322,A -85,B 0,C 180,E1 -6117.563,E2 -6117.563} C_VEL
LIN {X 0,Y 495.998,Z 429.326,A -85,B 0,C 180,E1 -6120,E2 -6120} C_VEL
LIN {X 0,Y 495.993,Z 429.32,A -85,B 0,C 180,E1 -6122.436,E2 -6122.436} C_VEL
LIN {X 0,Y 495.895,Z 429.334,A -85,B 0,C 180,E1 -6125.693,E2 -6125.693} C_VEL
LIN {X 0,Y 495.873,Z 429.34,A -85,B 0,C 180,E1 -6128.148,E2 -6128.148} C_VEL
LIN {X 0,Y 495.851,Z 429.341,A -85,B 0,C 180,E1 -6131.445,E2 -6131.445} C_VEL
LIN {X 0,Y 495.789,Z 429.347,A -85,B 0,C 180,E1 -6134.783,E2 -6134.783} C_VEL
LIN {X 0,Y 495.786,Z 429.351,A -85,B 0,C 180,E1 -6137.318,E2 -6137.318} C_VEL
LIN {X 0,Y 495.771,Z 429.356,A -85,B 0,C 180,E1 -6139.89,E2 -6139.89} C_VEL
LIN {X 0,Y 495.761,Z 429.351,A -85,B 0,C 180,E1 -6142.861,E2 -6142.861} C_VEL
LIN {X 0,Y 495.79,Z 429.351,A -85,B 0,C 180,E1 -6146.068,E2 -6146.068} C_VEL
LIN {X 0,Y 495.771,Z 429.349,A -85,B 0,C 180,E1 -6148.815,E2 -6148.815} C_VEL
LIN {X 0,Y 495.755,Z 429.359,A -85,B 0,C 180,E1 -6151.725,E2 -6151.725} C_VEL
LIN {X 0,Y 495.776,Z 429.35,A -85,B 0,C 180,E1 -6154.695,E2 -6154.695} C_VEL
LIN {X 0,Y 495.731,Z 429.362,A -85,B 0,C 180,E1 -6157.561,E2 -6157.561} C_VEL
LIN {X 0,Y 495.766,Z 429.351,A -85,B 0,C 180,E1 -6160.7,E2 -6160.7} C_VEL
LIN {X 0,Y 495.733,Z 429.36,A -85,B 0,C 180,E1 -6164.001,E2 -6164.001} C_VEL
LIN {X 0,Y 495.764,Z 429.353,A -85,B 0,C 180,E1 -6167.121,E2 -6167.121} C_VEL
LIN {X 0,Y 495.759,Z 429.359,A -85,B 0,C 180,E1 -6169.953,E2 -6169.953} C_VEL
LIN {X 0,Y 495.728,Z 429.356,A -85,B 0,C 180,E1 -6172.553,E2 -6172.553} C_VEL
LIN {X 0,Y 495.778,Z 429.356,A -85,B 0,C 180,E1 -6175.457,E2 -6175.457} C_VEL
LIN {X 0,Y 495.756,Z 429.358,A -85,B 0,C 180,E1 -6178.364,E2 -6178.364} C_VEL
LIN {X 0,Y 495.813,Z 429.422,A -85,B 0,C 180,E1 -6180.81,E2 -6180.81} C_VEL
LIN {X 0,Y 499.424,Z 444.666,A -85,B 0,C 180,E1 -6183.236,E2 -6183.236} C_VEL
LIN {X 0,Y 499.53,Z 449.392,A -85,B 0,C 180,E1 -6183.917,E2 -6183.917} C_VEL
LIN {X 0,Y 498.502,Z 471.38,A -85,B 0,C 180,E1 -6186.969,E2 -6186.969} C_VEL
LIN {X 0,Y 498.477,Z 473.851,A -85,B 0,C 180,E1 -6187.272,E2 -6187.272} C_VEL
LIN {X 0,Y 502.058,Z 491.721,A -85,B 0,C 180,E1 -6187.714,E2 -6187.714} C_VEL
LIN {X 0,Y 500.908,Z 626.701,A -85,B 0,C 180,E1 -6189.702,E2 -6189.702} C_VEL
LIN {X 0,Y 500.665,Z 643.992,A -85,B 0,C 180,E1 -6190.006,E2 -6190.006} C_VEL
LIN {X 0,Y 500.28,Z 658.821,A -85,B 0,C 180,E1 -6190.422,E2 -6190.422} C_VEL
LIN {X 0,Y 499.772,Z 673.292,A -85,B 0,C 180,E1 -6190.986,E2 -6190.986} C_VEL
LIN {X 0,Y 499.206,Z 686.325,A -85,B 0,C 180,E1 -6191.639,E2 -6191.639} C_VEL
LIN {X 0,Y 498.569,Z 699.585,A -85,B 0,C 180,E1 -6192.464,E2 -6192.464} C_VEL
LIN {X 0,Y 497.902,Z 713.078,A -85,B 0,C 180,E1 -6193.497,E2 -6193.497} C_VEL
LIN {X 0,Y 497.225,Z 725.363,A -85,B 0,C 180,E1 -6194.632,E2 -6194.632} C_VEL
LIN {X 0,Y 496.652,Z 736.578,A -85,B 0,C 180,E1 -6195.871,E2 -6195.871} C_VEL
LIN {X 0,Y 496.13,Z 747.463,A -85,B 0,C 180,E1 -6197.316,E2 -6197.316} C_VEL
LIN {X 0,Y 495.791,Z 756.527,A -85,B 0,C 180,E1 -6198.76,E2 -6198.76} C_VEL
LIN {X 0,Y 495.404,Z 764.04,A -85,B 0,C 180,E1 -6200.198,E2 -6200.198} C_VEL
LIN {X 0,Y 495.237,Z 771.057,A -85,B 0,C 180,E1 -6201.841,E2 -6201.841} C_VEL
LIN {X 0,Y 495.086,Z 776.811,A -85,B 0,C 180,E1 -6203.557,E2 -6203.557} C_VEL
LIN {X 0,Y 495.006,Z 780.741,A -85,B 0,C 180,E1 -6205.113,E2 -6205.113} C_VEL
LIN {X 0,Y 495.027,Z 783.665,A -85,B 0,C 180,E1 -6206.744,E2 -6206.744} C_VEL
LIN {X 0,Y 494.958,Z 785.406,A -85,B 0,C 180,E1 -6208.372,E2 -6208.372} C_VEL
LIN {X 0,Y 494.895,Z 786,A -85,B 0,C 180,E1 -6210,E2 -6210} C_VEL
LIN {X 0,Y 494.958,Z 785.401,A -85,B 0,C 180,E1 -6211.627,E2 -6211.627} C_VEL
LIN {X 0,Y 495.027,Z 783.654,A -85,B 0,C 180,E1 -6213.255,E2 -6213.255} C_VEL
LIN {X 0,Y 495.005,Z 780.729,A -85,B 0,C 180,E1 -6214.886,E2 -6214.886} C_VEL
LIN {X 0,Y 495.103,Z 776.562,A -85,B 0,C 180,E1 -6216.52,E2 -6216.52} C_VEL
LIN {X 0,Y 495.236,Z 771.038,A -85,B 0,C 180,E1 -6218.158,E2 -6218.158} C_VEL
LIN {X 0,Y 495.403,Z 764.008,A -85,B 0,C 180,E1 -6219.801,E2 -6219.801} C_VEL
LIN {X 0,Y 495.776,Z 756.49,A -85,B 0,C 180,E1 -6221.239,E2 -6221.239} C_VEL
LIN {X 0,Y 496.13,Z 747.422,A -85,B 0,C 180,E1 -6222.683,E2 -6222.683} C_VEL
LIN {X 0,Y 496.649,Z 736.526,A -85,B 0,C 180,E1 -6224.128,E2 -6224.128} C_VEL
LIN {X 0,Y 497.277,Z 724.275,A -85,B 0,C 180,E1 -6225.471,E2 -6225.471} C_VEL
LIN {X 0,Y 497.951,Z 711.784,A -85,B 0,C 180,E1 -6226.606,E2 -6226.606} C_VEL
LIN {X 0,Y 498.538,Z 699.5,A -85,B 0,C 180,E1 -6227.537,E2 -6227.537} C_VEL
LIN {X 0,Y 499.164,Z 686.224,A -85,B 0,C 180,E1 -6228.362,E2 -6228.362} C_VEL
LIN {X 0,Y 499.778,Z 672.111,A -85,B 0,C 180,E1 -6229.064,E2 -6229.064} C_VEL
LIN {X 0,Y 500.276,Z 657.34,A -85,B 0,C 180,E1 -6229.626,E2 -6229.626} C_VEL
LIN {X 0,Y 500.675,Z 642.543,A -85,B 0,C 180,E1 -6230.023,E2 -6230.023} C_VEL
LIN {X 0,Y 500.985,Z 619.697,A -85,B 0,C 180,E1 -6230.397,E2 -6230.397} C_VEL
LIN {X 0,Y 502.057,Z 491.956,A -85,B 0,C 180,E1 -6232.28,E2 -6232.28} C_VEL
LIN {X 0,Y 498.401,Z 473.116,A -85,B 0,C 180,E1 -6232.766,E2 -6232.766} C_VEL
LIN {X 0,Y 499.507,Z 449.175,A -85,B 0,C 180,E1 -6236.083,E2 -6236.083} C_VEL
LIN {X 0,Y 499.316,Z 444.448,A -85,B 0,C 180,E1 -6236.769,E2 -6236.769} C_VEL
LIN {X 0,Y 496.364,Z 431.788,A -85,B 0,C 180,E1 -6238.776,E2 -6238.776} C_VEL
LIN {X 0,Y 495.789,Z 429.357,A -85,B 0,C 180,E1 -6239.19,E2 -6239.19} C_VEL
LIN {X 0,Y 495.766,Z 429.358,A -85,B 0,C 180,E1 -6242.593,E2 -6242.593} C_VEL
LIN {X 0,Y 495.752,Z 429.354,A -85,B 0,C 180,E1 -6245.536,E2 -6245.536} C_VEL
LIN {X 0,Y 495.774,Z 429.353,A -85,B 0,C 180,E1 -6248.77,E2 -6248.77} C_VEL
LIN {X 0,Y 495.778,Z 429.354,A -85,B 0,C 180,E1 -6251.778,E2 -6251.778} C_VEL
LIN {X 0,Y 495.744,Z 429.356,A -85,B 0,C 180,E1 -6255.139,E2 -6255.139} C_VEL
LIN {X 0,Y 495.752,Z 429.359,A -85,B 0,C 180,E1 -6258.219,E2 -6258.219} C_VEL
LIN {X 0,Y 495.745,Z 429.354,A -85,B 0,C 180,E1 -6261.408,E2 -6261.408} C_VEL
LIN {X 0,Y 495.752,Z 429.358,A -85,B 0,C 180,E1 -6264.463,E2 -6264.463} C_VEL
LIN {X 0,Y 495.763,Z 429.35,A -85,B 0,C 180,E1 -6267.405,E2 -6267.405} C_VEL
LIN {X 0,Y 495.759,Z 429.357,A -85,B 0,C 180,E1 -6270.253,E2 -6270.253} C_VEL
LIN {X 0,Y 495.827,Z 429.342,A -85,B 0,C 180,E1 -6273.248,E2 -6273.248} C_VEL
LIN {X 0,Y 495.745,Z 429.354,A -85,B 0,C 180,E1 -6275.725,E2 -6275.725} C_VEL
LIN {X 0,Y 495.737,Z 429.361,A -85,B 0,C 180,E1 -6278.371,E2 -6278.371} C_VEL
LIN {X 0,Y 495.778,Z 429.351,A -85,B 0,C 180,E1 -6280.972,E2 -6280.972} C_VEL
LIN {X 0,Y 495.773,Z 429.347,A -85,B 0,C 180,E1 -6283.53,E2 -6283.53} C_VEL
LIN {X 0,Y 495.786,Z 429.353,A -85,B 0,C 180,E1 -6286.056,E2 -6286.056} C_VEL
LIN {X 0,Y 495.86,Z 429.345,A -85,B 0,C 180,E1 -6288.555,E2 -6288.555} C_VEL
LIN {X 0,Y 495.866,Z 429.34,A -85,B 0,C 180,E1 -6291.852,E2 -6291.852} C_VEL
LIN {X 0,Y 495.889,Z 429.34,A -85,B 0,C 180,E1 -6294.307,E2 -6294.307} C_VEL
LIN {X 0,Y 495.987,Z 429.322,A -85,B 0,C 180,E1 -6297.564,E2 -6297.564} C_VEL
LIN {X 0,Y 495.99,Z 429.327,A -85,B 0,C 180,E1 -6300,E2 -6300} C_VEL
LIN {X 0,Y 495.987,Z 429.33,A -85,B 0,C 180,E1 -6302.437,E2 -6302.437} C_VEL
LIN {X 0,Y 495.893,Z 429.335,A -85,B 0,C 180,E1 -6305.694,E2 -6305.694} C_VEL
LIN {X 0,Y 495.866,Z 429.343,A -85,B 0,C 180,E1 -6308.148,E2 -6308.148} C_VEL
LIN {X 0,Y 495.844,Z 429.34,A -85,B 0,C 180,E1 -6311.446,E2 -6311.446} C_VEL
LIN {X 0,Y 495.788,Z 429.352,A -85,B 0,C 180,E1 -6314.783,E2 -6314.783} C_VEL
LIN {X 0,Y 495.782,Z 429.349,A -85,B 0,C 180,E1 -6317.319,E2 -6317.319} C_VEL
LIN {X 0,Y 495.772,Z 429.352,A -85,B 0,C 180,E1 -6319.891,E2 -6319.891} C_VEL
LIN {X 0,Y 495.752,Z 429.357,A -85,B 0,C 180,E1 -6322.861,E2 -6322.861} C_VEL
LIN {X 0,Y 495.794,Z 429.353,A -85,B 0,C 180,E1 -6326.068,E2 -6326.068} C_VEL
LIN {X 0,Y 495.775,Z 429.354,A -85,B 0,C 180,E1 -6328.815,E2 -6328.815} C_VEL
LIN {X 0,Y 495.754,Z 429.355,A -85,B 0,C 180,E1 -6331.727,E2 -6331.727} C_VEL
LIN {X 0,Y 495.773,Z 429.355,A -85,B 0,C 180,E1 -6334.696,E2 -6334.696} C_VEL
LIN {X 0,Y 495.729,Z 429.359,A -85,B 0,C 180,E1 -6337.562,E2 -6337.562} C_VEL
LIN {X 0,Y 495.79,Z 429.354,A -85,B 0,C 180,E1 -6340.053,E2 -6340.053} C_VEL
LIN {X 0,Y 495.813,Z 429.479,A -85,B 0,C 180,E1 -6342.178,E2 -6342.178} C_VEL
LIN {X 0,Y 498.436,Z 441.278,A -85,B 0,C 180,E1 -6344.288,E2 -6344.288} C_VEL
LIN {X 0,Y 498.402,Z 447.524,A -85,B 0,C 180,E1 -6345.309,E2 -6345.309} C_VEL
LIN {X 0,Y 502.256,Z 464.573,A -85,B 0,C 180,E1 -6345.768,E2 -6345.768} C_VEL
LIN {X 0,Y 501.33,Z 560.128,A -85,B 0,C 180,E1 -6347.177,E2 -6347.177} C_VEL
LIN {X 0,Y 500.67,Z 565.976,A -85,B 0,C 180,E1 -6347.236,E2 -6347.236} C_VEL
LIN {X 0,Y 495.118,Z 585.024,A -85,B 0,C 180,E1 -6347.281,E2 -6347.281} C_VEL
LIN {X 0,Y 494.44,Z 590.873,A -85,B 0,C 180,E1 -6347.341,E2 -6347.341} C_VEL
LIN {X 0,Y 494.125,Z 614.91,A -85,B 0,C 180,E1 -6347.736,E2 -6347.736} C_VEL
LIN {X 0,Y 493.731,Z 630.01,A -85,B 0,C 180,E1 -6348.147,E2 -6348.147} C_VEL
LIN {X 0,Y 493.254,Z 644.595,A -85,B 0,C 180,E1 -6348.711,E2 -6348.711} C_VEL
LIN {X 0,Y 492.651,Z 658.185,A -85,B 0,C 180,E1 -6349.394,E2 -6349.394} C_VEL
LIN {X 0,Y 491.923,Z 672.541,A -85,B 0,C 180,E1 -6350.307,E2 -6350.307} C_VEL
LIN {X 0,Y 491.249,Z 684.714,A -85,B 0,C 180,E1 -6351.253,E2 -6351.253} C_VEL
LIN {X 0,Y 490.534,Z 697.798,A -85,B 0,C 180,E1 -6352.491,E2 -6352.491} C_VEL
LIN {X 0,Y 489.858,Z 709.123,A -85,B 0,C 180,E1 -6353.781,E2 -6353.781} C_VEL
LIN {X 0,Y 489.322,Z 719.409,A -85,B 0,C 180,E1 -6355.187,E2 -6355.187} C_VEL
LIN {X 0,Y 488.846,Z 728.56,A -85,B 0,C 180,E1 -6356.69,E2 -6356.69} C_VEL
LIN {X 0,Y 488.48,Z 735.644,A -85,B 0,C 180,E1 -6358.089,E2 -6358.089} C_VEL
LIN {X 0,Y 488.256,Z 742.546,A -85,B 0,C 180,E1 -6359.75,E2 -6359.75} C_VEL
LIN {X 0,Y 488.013,Z 748.135,A -85,B 0,C 180,E1 -6361.46,E2 -6361.46} C_VEL
LIN {X 0,Y 487.983,Z 750.996,A -85,B 0,C 180,E1 -6362.558,E2 -6362.558} C_VEL
LIN {X 0,Y 487.802,Z 754.526,A -85,B 0,C 180,E1 -6364.392,E2 -6364.392} C_VEL
LIN {X 0,Y 487.825,Z 755.739,A -85,B 0,C 180,E1 -6365.305,E2 -6365.305} C_VEL
LIN {X 0,Y 487.76,Z 757.112,A -85,B 0,C 180,E1 -6367.106,E2 -6367.106} C_VEL
LIN {X 0,Y 487.769,Z 757.137,A -85,B 0,C 180,E1 -6368.888,E2 -6368.888} C_VEL
LIN {X 0,Y 487.802,Z 755.866,A -85,B 0,C 180,E1 -6370.649,E2 -6370.649} C_VEL
LIN {X 0,Y 487.87,Z 753.323,A -85,B 0,C 180,E1 -6372.392,E2 -6372.392} C_VEL
LIN {X 0,Y 488.03,Z 749.481,A -85,B 0,C 180,E1 -6374.121,E2 -6374.121} C_VEL
LIN {X 0,Y 488.182,Z 744.305,A -85,B 0,C 180,E1 -6375.834,E2 -6375.834} C_VEL
LIN {X 0,Y 488.412,Z 737.683,A -85,B 0,C 180,E1 -6377.536,E2 -6377.536} C_VEL
LIN {X 0,Y 488.751,Z 730.551,A -85,B 0,C 180,E1 -6379.017,E2 -6379.017} C_VEL
LIN {X 0,Y 489.152,Z 722.018,A -85,B 0,C 180,E1 -6380.49,E2 -6380.49} C_VEL
LIN {X 0,Y 489.722,Z 711.59,A -85,B 0,C 180,E1 -6381.982,E2 -6381.982} C_VEL
LIN {X 0,Y 490.319,Z 701.344,A -85,B 0,C 180,E1 -6383.209,E2 -6383.209} C_VEL
LIN {X 0,Y 490.946,Z 690.048,A -85,B 0,C 180,E1 -6384.352,E2 -6384.352} C_VEL
LIN {X 0,Y 491.613,Z 677.828,A -85,B 0,C 180,E1 -6385.388,E2 -6385.388} C_VEL
LIN {X 0,Y 492.364,Z 664.457,A -85,B 0,C 180,E1 -6386.318,E2 -6386.318} C_VEL
LIN {X 0,Y 492.99,Z 651.032,A -85,B 0,C 180,E1 -6387.071,E2 -6387.071} C_VEL
LIN {X 0,Y 493.524,Z 636.623,A -85,B 0,C 180,E1 -6387.705,E2 -6387.705} C_VEL
LIN {X 0,Y 493.974,Z 621.575,A -85,B 0,C 180,E1 -6388.192,E2 -6388.192} C_VEL
LIN {X 0,Y 494.238,Z 605.917,A -85,B 0,C 180,E1 -6388.524,E2 -6388.524} C_VEL
LIN {X 0,Y 495.599,Z 464.947,A -85,B 0,C 180,E1 -6390.631,E2 -6390.631} C_VEL
LIN {X 0,Y 491.606,Z 447.45,A -85,B 0,C 180,E1 -6391.121,E2 -6391.121} C_VEL
LIN {X 0,Y 491.583,Z 443.083,A -85,B 0,C 180,E1 -6391.844,E2 -6391.844} C_VEL
LIN {X 0,Y 489.638,Z 433.844,A -85,B 0,C 180,E1 -6393.498,E2 -6393.498} C_VEL
LIN {X 0,Y 488.727,Z 430.235,A -85,B 0,C 180,E1 -6394.175,E2 -6394.175} C_VEL
LIN {X 0,Y 488.795,Z 430.223,A -85,B 0,C 180,E1 -6396.605,E2 -6396.605} C_VEL
LIN {X 0,Y 488.788,Z 430.225,A -85,B 0,C 180,E1 -6399.101,E2 -6399.101} C_VEL
LIN {X 0,Y 488.827,Z 430.22,A -85,B 0,C 180,E1 -6402.134,E2 -6402.134} C_VEL
LIN {X 0,Y 488.781,Z 430.227,A -85,B 0,C 180,E1 -6405.555,E2 -6405.555} C_VEL
LIN {X 0,Y 488.759,Z 430.224,A -85,B 0,C 180,E1 -6408.442,E2 -6408.442} C_VEL
LIN {X 0,Y 488.712,Z 430.231,A -85,B 0,C 180,E1 -6411.071,E2 -6411.071} C_VEL
LIN {X 0,Y 488.698,Z 430.235,A -85,B 0,C 180,E1 -6413.745,E2 -6413.745} C_VEL
LIN {X 0,Y 488.796,Z 430.22,A -85,B 0,C 180,E1 -6416.944,E2 -6416.944} C_VEL
LIN {X 0,Y 488.714,Z 430.231,A -85,B 0,C 180,E1 -6420.363,E2 -6420.363} C_VEL
LIN {X 0,Y 488.739,Z 430.227,A -85,B 0,C 180,E1 -6423.484,E2 -6423.484} C_VEL
LIN {X 0,Y 488.691,Z 430.231,A -85,B 0,C 180,E1 -6426.355,E2 -6426.355} C_VEL
LIN {X 0,Y 488.704,Z 430.229,A -85,B 0,C 180,E1 -6429.254,E2 -6429.254} C_VEL
LIN {X 0,Y 488.727,Z 430.235,A -85,B 0,C 180,E1 -6431.602,E2 -6431.602} C_VEL
LIN {X 0,Y 488.715,Z 430.228,A -85,B 0,C 180,E1 -6434.801,E2 -6434.801} C_VEL
LIN {X 0,Y 488.694,Z 430.237,A -85,B 0,C 180,E1 -6437.474,E2 -6437.474} C_VEL
LIN {X 0,Y 488.735,Z 430.231,A -85,B 0,C 180,E1 -6439.676,E2 -6439.676} C_VEL
LIN {X 0,Y 488.682,Z 430.233,A -85,B 0,C 180,E1 -6442.277,E2 -6442.277} C_VEL
LIN {X 0,Y 488.73,Z 430.224,A -85,B 0,C 180,E1 -6445.051,E2 -6445.051} C_VEL
LIN {X 0,Y 488.705,Z 430.232,A -85,B 0,C 180,E1 -6448.046,E2 -6448.046} C_VEL
LIN {X 0,Y 488.724,Z 430.223,A -85,B 0,C 180,E1 -6450.729,E2 -6450.729} C_VEL
LIN {X 0,Y 488.768,Z 430.229,A -85,B 0,C 180,E1 -6453.528,E2 -6453.528} C_VEL
LIN {X 0,Y 488.689,Z 430.226,A -85,B 0,C 180,E1 -6456.254,E2 -6456.254} C_VEL
LIN {X 0,Y 488.747,Z 430.226,A -85,B 0,C 180,E1 -6459.175,E2 -6459.175} C_VEL
LIN {X 0,Y 488.734,Z 430.222,A -85,B 0,C 180,E1 -6462.423,E2 -6462.423} C_VEL
LIN {X 0,Y 488.762,Z 430.22,A -85,B 0,C 180,E1 -6464.999,E2 -6464.999} C_VEL
LIN {X 0,Y 488.805,Z 430.216,A -85,B 0,C 180,E1 -6468.387,E2 -6468.387} C_VEL
LIN {X 0,Y 488.817,Z 430.22,A -85,B 0,C 180,E1 -6471.733,E2 -6471.733} C_VEL
LIN {X 0,Y 488.855,Z 430.213,A -85,B 0,C 180,E1 -6474.224,E2 -6474.224} C_VEL
LIN {X 0,Y 488.961,Z 430.198,A -85,B 0,C 180,E1 -6477.528,E2 -6477.528} C_VEL
LIN {X 0,Y 488.954,Z 430.199,A -85,B 0,C 180,E1 -6480.823,E2 -6480.823} C_VEL
LIN {X 0,Y 488.961,Z 430.196,A -85,B 0,C 180,E1 -6482.471,E2 -6482.471} C_VEL
LIN {X 0,Y 488.854,Z 430.212,A -85,B 0,C 180,E1 -6485.776,E2 -6485.776} C_VEL
LIN {X 0,Y 488.817,Z 430.218,A -85,B 0,C 180,E1 -6488.266,E2 -6488.266} C_VEL
LIN {X 0,Y 488.805,Z 430.217,A -85,B 0,C 180,E1 -6491.612,E2 -6491.612} C_VEL
LIN {X 0,Y 488.761,Z 430.224,A -85,B 0,C 180,E1 -6495,E2 -6495} C_VEL
LIN {X 0,Y 488.754,Z 430.217,A -85,B 0,C 180,E1 -6498.442,E2 -6498.442} C_VEL
LIN {X 0,Y 488.706,Z 430.231,A -85,B 0,C 180,E1 -6501.071,E2 -6501.071} C_VEL
LIN {X 0,Y 488.693,Z 430.239,A -85,B 0,C 180,E1 -6503.745,E2 -6503.745} C_VEL
LIN {X 0,Y 488.791,Z 430.22,A -85,B 0,C 180,E1 -6506.944,E2 -6506.944} C_VEL
LIN {X 0,Y 488.709,Z 430.23,A -85,B 0,C 180,E1 -6510.363,E2 -6510.363} C_VEL
LIN {X 0,Y 488.735,Z 430.232,A -85,B 0,C 180,E1 -6513.484,E2 -6513.484} C_VEL
LIN {X 0,Y 488.689,Z 430.234,A -85,B 0,C 180,E1 -6516.356,E2 -6516.356} C_VEL
LIN {X 0,Y 488.701,Z 430.234,A -85,B 0,C 180,E1 -6519.254,E2 -6519.254} C_VEL
LIN {X 0,Y 488.707,Z 430.237,A -85,B 0,C 180,E1 -6521.6,E2 -6521.6} C_VEL
LIN {X 0,Y 488.712,Z 430.23,A -85,B 0,C 180,E1 -6524.801,E2 -6524.801} C_VEL
LIN {X 0,Y 488.735,Z 430.233,A -85,B 0,C 180,E1 -6527.479,E2 -6527.479} C_VEL
LIN {X 0,Y 488.701,Z 430.232,A -85,B 0,C 180,E1 -6530.746,E2 -6530.746} C_VEL
LIN {X 0,Y 488.677,Z 430.24,A -85,B 0,C 180,E1 -6533.868,E2 -6533.868} C_VEL
LIN {X 0,Y 488.739,Z 430.231,A -85,B 0,C 180,E1 -6536.877,E2 -6536.877} C_VEL
LIN {X 0,Y 488.758,Z 430.302,A -85,B 0,C 180,E1 -6540.51,E2 -6540.51} C_VEL
LIN {X 0,Y 492.507,Z 446.042,A -85,B 0,C 180,E1 -6543.059,E2 -6543.059} C_VEL
LIN {X 0,Y 492.758,Z 449.195,A -85,B 0,C 180,E1 -6543.531,E2 -6543.531} C_VEL
LIN {X 0,Y 491.704,Z 471.184,A -85,B 0,C 180,E1 -6546.632,E2 -6546.632} C_VEL
LIN {X 0,Y 491.652,Z 473.657,A -85,B 0,C 180,E1 -6546.94,E2 -6546.94} C_VEL
LIN {X 0,Y 495.514,Z 493.169,A -85,B 0,C 180,E1 -6547.429,E2 -6547.429} C_VEL
LIN {X 0,Y 494.111,Z 639.609,A -85,B 0,C 180,E1 -6549.633,E2 -6549.633} C_VEL
LIN {X 0,Y 493.631,Z 655.548,A -85,B 0,C 180,E1 -6550.04,E2 -6550.04} C_VEL
LIN {X 0,Y 493.13,Z 670.269,A -85,B 0,C 180,E1 -6550.588,E2 -6550.588} C_VEL
LIN {X 0,Y 492.501,Z 684.243,A -85,B 0,C 180,E1 -6551.272,E2 -6551.272} C_VEL
LIN {X 0,Y 491.842,Z 697.815,A -85,B 0,C 180,E1 -6552.108,E2 -6552.108} C_VEL
LIN {X 0,Y 491.143,Z 710.321,A -85,B 0,C 180,E1 -6553.049,E2 -6553.049} C_VEL
LIN {X 0,Y 490.451,Z 723.033,A -85,B 0,C 180,E1 -6554.201,E2 -6554.201} C_VEL
LIN {X 0,Y 489.789,Z 734.58,A -85,B 0,C 180,E1 -6555.457,E2 -6555.457} C_VEL
LIN {X 0,Y 489.274,Z 744.3,A -85,B 0,C 180,E1 -6556.713,E2 -6556.713} C_VEL
LIN {X 0,Y 488.781,Z 754.027,A -85,B 0,C 180,E1 -6558.207,E2 -6558.207} C_VEL
LIN {X 0,Y 488.483,Z 761.799,A -85,B 0,C 180,E1 -6559.639,E2 -6559.639} C_VEL
LIN {X 0,Y 488.198,Z 769.222,A -85,B 0,C 180,E1 -6561.306,E2 -6561.306} C_VEL
LIN {X 0,Y 488.068,Z 775.112,A -85,B 0,C 180,E1 -6562.969,E2 -6562.969} C_VEL
LIN {X 0,Y 487.995,Z 778.611,A -85,B 0,C 180,E1 -6564.214,E2 -6564.214} C_VEL
LIN {X 0,Y 487.89,Z 782.146,A -85,B 0,C 180,E1 -6565.869,E2 -6565.869} C_VEL
LIN {X 0,Y 487.882,Z 784.473,A -85,B 0,C 180,E1 -6567.523,E2 -6567.523} C_VEL
LIN {X 0,Y 487.831,Z 785.641,A -85,B 0,C 180,E1 -6569.174,E2 -6569.174} C_VEL
LIN {X 0,Y 487.831,Z 785.638,A -85,B 0,C 180,E1 -6570.825,E2 -6570.825} C_VEL
LIN {X 0,Y 487.882,Z 784.462,A -85,B 0,C 180,E1 -6572.476,E2 -6572.476} C_VEL
LIN {X 0,Y 487.89,Z 782.13,A -85,B 0,C 180,E1 -6574.13,E2 -6574.13} C_VEL
LIN {X 0,Y 487.994,Z 778.595,A -85,B 0,C 180,E1 -6575.785,E2 -6575.785} C_VEL
LIN {X 0,Y 488.069,Z 773.762,A -85,B 0,C 180,E1 -6577.446,E2 -6577.446} C_VEL
LIN {X 0,Y 488.262,Z 767.504,A -85,B 0,C 180,E1 -6579.11,E2 -6579.11} C_VEL
LIN {X 0,Y 488.608,Z 759.646,A -85,B 0,C 180,E1 -6580.776,E2 -6580.776} C_VEL
LIN {X 0,Y 488.836,Z 751.911,A -85,B 0,C 180,E1 -6582.141,E2 -6582.141} C_VEL
LIN {X 0,Y 489.346,Z 742.747,A -85,B 0,C 180,E1 -6583.496,E2 -6583.496} C_VEL
LIN {X 0,Y 489.862,Z 732.719,A -85,B 0,C 180,E1 -6584.753,E2 -6584.753} C_VEL
LIN {X 0,Y 490.51,Z 721.748,A -85,B 0,C 180,E1 -6585.917,E2 -6585.917} C_VEL
LIN {X 0,Y 491.174,Z 708.94,A -85,B 0,C 180,E1 -6587.056,E2 -6587.056} C_VEL
LIN {X 0,Y 491.934,Z 696.122,A -85,B 0,C 180,E1 -6587.995,E2 -6587.995} C_VEL
LIN {X 0,Y 492.57,Z 682.128,A -85,B 0,C 180,E1 -6588.832,E2 -6588.832} C_VEL
LIN {X 0,Y 493.197,Z 667.91,A -85,B 0,C 180,E1 -6589.502,E2 -6589.502} C_VEL
LIN {X 0,Y 493.682,Z 653.317,A -85,B 0,C 180,E1 -6590.021,E2 -6590.021} C_VEL
LIN {X 0,Y 494.062,Z 637.989,A -85,B 0,C 180,E1 -6590.395,E2 -6590.395} C_VEL
LIN {X 0,Y 495.552,Z 493.357,A -85,B 0,C 180,E1 -6592.563,E2 -6592.563} C_VEL
LIN {X 0,Y 491.552,Z 472.891,A -85,B 0,C 180,E1 -6593.101,E2 -6593.101} C_VEL
LIN {X 0,Y 492.689,Z 450.544,A -85,B 0,C 180,E1 -6596.244,E2 -6596.244} C_VEL
LIN {X 0,Y 492.7,Z 447.397,A -85,B 0,C 180,E1 -6596.699,E2 -6596.699} C_VEL
LIN {X 0,Y 490.086,Z 435.723,A -85,B 0,C 180,E1 -6598.568,E2 -6598.568} C_VEL
LIN {X 0,Y 488.735,Z 430.236,A -85,B 0,C 180,E1 -6599.505,E2 -6599.505} C_VEL
LIN {X 0,Y 488.736,Z 430.229,A -85,B 0,C 180,E1 -6603.122,E2 -6603.122} C_VEL
LIN {X 0,Y 488.68,Z 430.24,A -85,B 0,C 180,E1 -6606.131,E2 -6606.131} C_VEL
LIN {X 0,Y 488.744,Z 430.227,A -85,B 0,C 180,E1 -6609.249,E2 -6609.249} C_VEL
LIN {X 0,Y 488.727,Z 430.23,A -85,B 0,C 180,E1 -6612.521,E2 -6612.521} C_VEL
LIN {X 0,Y 488.706,Z 430.232,A -85,B 0,C 180,E1 -6615.198,E2 -6615.198} C_VEL
LIN {X 0,Y 488.703,Z 430.239,A -85,B 0,C 180,E1 -6618.399,E2 -6618.399} C_VEL
LIN {X 0,Y 488.698,Z 430.233,A -85,B 0,C 180,E1 -6620.947,E2 -6620.947} C_VEL
LIN {X 0,Y 488.679,Z 430.237,A -85,B 0,C 180,E1 -6623.868,E2 -6623.868} C_VEL
LIN {X 0,Y 488.733,Z 430.227,A -85,B 0,C 180,E1 -6626.877,E2 -6626.877} C_VEL
LIN {X 0,Y 488.717,Z 430.23,A -85,B 0,C 180,E1 -6629.78,E2 -6629.78} C_VEL
LIN {X 0,Y 488.792,Z 430.219,A -85,B 0,C 180,E1 -6633.054,E2 -6633.054} C_VEL
LIN {X 0,Y 488.686,Z 430.237,A -85,B 0,C 180,E1 -6636.254,E2 -6636.254} C_VEL
LIN {X 0,Y 488.738,Z 430.224,A -85,B 0,C 180,E1 -6639.175,E2 -6639.175} C_VEL
LIN {X 0,Y 488.751,Z 430.226,A -85,B 0,C 180,E1 -6641.628,E2 -6641.628} C_VEL
LIN {X 0,Y 488.754,Z 430.225,A -85,B 0,C 180,E1 -6645,E2 -6645} C_VEL
LIN {X 0,Y 488.822,Z 430.224,A -85,B 0,C 180,E1 -6648.388,E2 -6648.388} C_VEL
LIN {X 0,Y 488.811,Z 430.218,A -85,B 0,C 180,E1 -6651.734,E2 -6651.734} C_VEL
LIN {X 0,Y 488.848,Z 430.216,A -85,B 0,C 180,E1 -6654.224,E2 -6654.224} C_VEL
LIN {X 0,Y 488.955,Z 430.197,A -85,B 0,C 180,E1 -6657.529,E2 -6657.529} C_VEL
LIN {X 0,Y 488.948,Z 430.2,A -85,B 0,C 180,E1 -6660.824,E2 -6660.824} C_VEL
LIN {X 0,Y 488.955,Z 430.207,A -85,B 0,C 180,E1 -6662.472,E2 -6662.472} C_VEL
LIN {X 0,Y 488.852,Z 430.212,A -85,B 0,C 180,E1 -6665.776,E2 -6665.776} C_VEL
LIN {X 0,Y 488.811,Z 430.222,A -85,B 0,C 180,E1 -6668.267,E2 -6668.267} C_VEL
LIN {X 0,Y 488.798,Z 430.218,A -85,B 0,C 180,E1 -6671.613,E2 -6671.613} C_VEL
LIN {X 0,Y 488.758,Z 430.226,A -85,B 0,C 180,E1 -6675.001,E2 -6675.001} C_VEL
LIN {X 0,Y 488.748,Z 430.232,A -85,B 0,C 180,E1 -6678.443,E2 -6678.443} C_VEL
LIN {X 0,Y 488.702,Z 430.232,A -85,B 0,C 180,E1 -6681.071,E2 -6681.071} C_VEL
LIN {X 0,Y 488.688,Z 430.235,A -85,B 0,C 180,E1 -6683.746,E2 -6683.746} C_VEL
LIN {X 0,Y 488.793,Z 430.223,A -85,B 0,C 180,E1 -6686.946,E2 -6686.946} C_VEL
LIN {X 0,Y 488.714,Z 430.233,A -85,B 0,C 180,E1 -6690.366,E2 -6690.366} C_VEL
LIN {X 0,Y 488.731,Z 430.229,A -85,B 0,C 180,E1 -6693.485,E2 -6693.485} C_VEL
LIN {X 0,Y 488.686,Z 430.241,A -85,B 0,C 180,E1 -6696.357,E2 -6696.357} C_VEL
LIN {X 0,Y 488.745,Z 430.231,A -85,B 0,C 180,E1 -6699.25,E2 -6699.25} C_VEL
LIN {X 0,Y 488.793,Z 430.409,A -85,B 0,C 180,E1 -6701.897,E2 -6701.897} C_VEL
LIN {X 0,Y 491.646,Z 443.301,A -85,B 0,C 180,E1 -6704.242,E2 -6704.242} C_VEL
LIN {X 0,Y 491.606,Z 447.718,A -85,B 0,C 180,E1 -6704.972,E2 -6704.972} C_VEL
LIN {X 0,Y 495.672,Z 465.534,A -85,B 0,C 180,E1 -6705.466,E2 -6705.466} C_VEL
LIN {X 0,Y 494.44,Z 590.873,A -85,B 0,C 180,E1 -6707.341,E2 -6707.341} C_VEL
LIN {X 0,Y 493.772,Z 596.73,A -85,B 0,C 180,E1 -6707.398,E2 -6707.398} C_VEL
LIN {X 0,Y 488.135,Z 615.738,A -85,B 0,C 180,E1 -6707.482,E2 -6707.482} C_VEL
LIN {X 0,Y 487.332,Z 621.495,A -85,B 0,C 180,E1 -6707.6,E2 -6707.6} C_VEL
LIN {X 0,Y 486.869,Z 635.538,A -85,B 0,C 180,E1 -6708.048,E2 -6708.048} C_VEL
LIN {X 0,Y 486.295,Z 650.866,A -85,B 0,C 180,E1 -6708.722,E2 -6708.722} C_VEL
LIN {X 0,Y 485.622,Z 664.37,A -85,B 0,C 180,E1 -6709.486,E2 -6709.486} C_VEL
LIN {X 0,Y 484.846,Z 678.812,A -85,B 0,C 180,E1 -6710.508,E2 -6710.508} C_VEL
LIN {X 0,Y 484.045,Z 691.733,A -85,B 0,C 180,E1 -6711.633,E2 -6711.633} C_VEL
LIN {X 0,Y 483.38,Z 702.906,A -85,B 0,C 180,E1 -6712.802,E2 -6712.802} C_VEL
LIN {X 0,Y 482.686,Z 713.533,A -85,B 0,C 180,E1 -6714.124,E2 -6714.124} C_VEL
LIN {X 0,Y 482.09,Z 723.423,A -85,B 0,C 180,E1 -6715.597,E2 -6715.597} C_VEL
LIN {X 0,Y 481.717,Z 731.684,A -85,B 0,C 180,E1 -6717.082,E2 -6717.082} C_VEL
LIN {X 0,Y 481.345,Z 738.441,A -85,B 0,C 180,E1 -6718.536,E2 -6718.536} C_VEL
LIN {X 0,Y 481.1,Z 744.813,A -85,B 0,C 180,E1 -6720.22,E2 -6720.22} C_VEL
LIN {X 0,Y 480.911,Z 749.227,A -85,B 0,C 180,E1 -6721.683,E2 -6721.683} C_VEL
LIN {X 0,Y 480.858,Z 752.454,A -85,B 0,C 180,E1 -6723.069,E2 -6723.069} C_VEL
LIN {X 0,Y 480.72,Z 755.633,A -85,B 0,C 180,E1 -6725.017,E2 -6725.017} C_VEL
LIN {X 0,Y 480.676,Z 757.32,A -85,B 0,C 180,E1 -6727.092,E2 -6727.092} C_VEL
LIN {X 0,Y 480.67,Z 757.409,A -85,B 0,C 180,E1 -6728.56,E2 -6728.56} C_VEL
LIN {X 0,Y 480.696,Z 756.391,A -85,B 0,C 180,E1 -6730.351,E2 -6730.351} C_VEL
LIN {X 0,Y 480.791,Z 754.098,A -85,B 0,C 180,E1 -6732.124,E2 -6732.124} C_VEL
LIN {X 0,Y 480.925,Z 750.516,A -85,B 0,C 180,E1 -6733.88,E2 -6733.88} C_VEL
LIN {X 0,Y 481.087,Z 745.605,A -85,B 0,C 180,E1 -6735.621,E2 -6735.621} C_VEL
LIN {X 0,Y 481.306,Z 739.273,A -85,B 0,C 180,E1 -6737.349,E2 -6737.349} C_VEL
LIN {X 0,Y 481.665,Z 732.447,A -85,B 0,C 180,E1 -6738.853,E2 -6738.853} C_VEL
LIN {X 0,Y 482.043,Z 724.237,A -85,B 0,C 180,E1 -6740.348,E2 -6740.348} C_VEL
LIN {X 0,Y 482.586,Z 714.803,A -85,B 0,C 180,E1 -6741.78,E2 -6741.78} C_VEL
LIN {X 0,Y 483.285,Z 704.335,A -85,B 0,C 180,E1 -6743.11,E2 -6743.11} C_VEL
LIN {X 0,Y 483.963,Z 692.463,A -85,B 0,C 180,E1 -6744.375,E2 -6744.375} C_VEL
LIN {X 0,Y 484.755,Z 679.338,A -85,B 0,C 180,E1 -6745.531,E2 -6745.531} C_VEL
LIN {X 0,Y 485.537,Z 666.231,A -85,B 0,C 180,E1 -6746.474,E2 -6746.474} C_VEL
LIN {X 0,Y 486.179,Z 653.043,A -85,B 0,C 180,E1 -6747.245,E2 -6747.245} C_VEL
LIN {X 0,Y 486.745,Z 639.356,A -85,B 0,C 180,E1 -6747.88,E2 -6747.88} C_VEL
LIN {X 0,Y 487.223,Z 624.455,A -85,B 0,C 180,E1 -6748.399,E2 -6748.399} C_VEL
LIN {X 0,Y 487.564,Z 608.943,A -85,B 0,C 180,E1 -6748.762,E2 -6748.762} C_VEL
LIN {X 0,Y 489.043,Z 465.974,A -85,B 0,C 180,E1 -6750.937,E2 -6750.937} C_VEL
LIN {X 0,Y 484.821,Z 447.67,A -85,B 0,C 180,E1 -6751.454,E2 -6751.454} C_VEL
LIN {X 0,Y 484.605,Z 444.019,A -85,B 0,C 180,E1 -6752.078,E2 -6752.078} C_VEL
LIN {X 0,Y 482.582,Z 434.834,A -85,B 0,C 180,E1 -6753.758,E2 -6753.758} C_VEL
LIN {X 0,Y 481.725,Z 431.106,A -85,B 0,C 180,E1 -6754.472,E2 -6754.472} C_VEL
LIN {X 0,Y 481.779,Z 431.099,A -85,B 0,C 180,E1 -6757.27,E2 -6757.27} C_VEL
LIN {X 0,Y 481.723,Z 431.099,A -85,B 0,C 180,E1 -6760.083,E2 -6760.083} C_VEL
LIN {X 0,Y 481.745,Z 431.1,A -85,B 0,C 180,E1 -6762.641,E2 -6762.641} C_VEL
LIN {X 0,Y 481.73,Z 431.105,A -85,B 0,C 180,E1 -6765.659,E2 -6765.659} C_VEL
LIN {X 0,Y 481.716,Z 431.101,A -85,B 0,C 180,E1 -6768.722,E2 -6768.722} C_VEL
LIN {X 0,Y 481.652,Z 431.113,A -85,B 0,C 180,E1 -6771.395,E2 -6771.395} C_VEL
LIN {X 0,Y 481.682,Z 431.105,A -85,B 0,C 180,E1 -6774.113,E2 -6774.113} C_VEL
LIN {X 0,Y 481.751,Z 431.099,A -85,B 0,C 180,E1 -6777.139,E2 -6777.139} C_VEL
LIN {X 0,Y 481.683,Z 431.113,A -85,B 0,C 180,E1 -6779.741,E2 -6779.741} C_VEL
LIN {X 0,Y 481.677,Z 431.1,A -85,B 0,C 180,E1 -6782.674,E2 -6782.674} C_VEL
LIN {X 0,Y 481.645,Z 431.117,A -85,B 0,C 180,E1 -6785.709,E2 -6785.709} C_VEL
LIN {X 0,Y 481.674,Z 431.102,A -85,B 0,C 180,E1 -6788.859,E2 -6788.859} C_VEL
LIN {X 0,Y 481.665,Z 431.11,A -85,B 0,C 180,E1 -6791.914,E2 -6791.914} C_VEL
LIN {X 0,Y 481.663,Z 431.107,A -85,B 0,C 180,E1 -6794.457,E2 -6794.457} C_VEL
LIN {X 0,Y 481.651,Z 431.109,A -85,B 0,C 180,E1 -6797.839,E2 -6797.839} C_VEL
LIN {X 0,Y 481.716,Z 431.101,A -85,B 0,C 180,E1 -6800.646,E2 -6800.646} C_VEL
LIN {X 0,Y 481.645,Z 431.107,A -85,B 0,C 180,E1 -6804.291,E2 -6804.291} C_VEL
LIN {X 0,Y 481.673,Z 431.11,A -85,B 0,C 180,E1 -6807.326,E2 -6807.326} C_VEL
LIN {X 0,Y 481.68,Z 431.101,A -85,B 0,C 180,E1 -6810.259,E2 -6810.259} C_VEL
LIN {X 0,Y 481.754,Z 431.098,A -85,B 0,C 180,E1 -6813.112,E2 -6813.112} C_VEL
LIN {X 0,Y 481.675,Z 431.103,A -85,B 0,C 180,E1 -6815.886,E2 -6815.886} C_VEL
LIN {X 0,Y 481.703,Z 431.102,A -85,B 0,C 180,E1 -6819.027,E2 -6819.027} C_VEL
LIN {X 0,Y 481.707,Z 431.099,A -85,B 0,C 180,E1 -6822.158,E2 -6822.158} C_VEL
LIN {X 0,Y 481.743,Z 431.094,A -85,B 0,C 180,E1 -6824.776,E2 -6824.776} C_VEL
LIN {X 0,Y 481.751,Z 431.096,A -85,B 0,C 180,E1 -6828.215,E2 -6828.215} C_VEL
LIN {X 0,Y 481.763,Z 431.096,A -85,B 0,C 180,E1 -6831.611,E2 -6831.611} C_VEL
LIN {X 0,Y 481.816,Z 431.09,A -85,B 0,C 180,E1 -6834.139,E2 -6834.139} C_VEL
LIN {X 0,Y 481.928,Z 431.073,A -85,B 0,C 180,E1 -6837.492,E2 -6837.492} C_VEL
LIN {X 0,Y 481.905,Z 431.078,A -85,B 0,C 180,E1 -6840.835,E2 -6840.835} C_VEL
LIN {X 0,Y 481.928,Z 431.071,A -85,B 0,C 180,E1 -6842.507,E2 -6842.507} C_VEL
LIN {X 0,Y 481.815,Z 431.09,A -85,B 0,C 180,E1 -6845.86,E2 -6845.86} C_VEL
LIN {X 0,Y 481.763,Z 431.096,A -85,B 0,C 180,E1 -6848.388,E2 -6848.388} C_VEL
LIN {X 0,Y 481.75,Z 431.094,A -85,B 0,C 180,E1 -6851.785,E2 -6851.785} C_VEL
LIN {X 0,Y 481.742,Z 431.1,A -85,B 0,C 180,E1 -6855.224,E2 -6855.224} C_VEL
LIN {X 0,Y 481.711,Z 431.094,A -85,B 0,C 180,E1 -6858.722,E2 -6858.722} C_VEL
LIN {X 0,Y 481.645,Z 431.114,A -85,B 0,C 180,E1 -6861.395,E2 -6861.395} C_VEL
LIN {X 0,Y 481.677,Z 431.109,A -85,B 0,C 180,E1 -6864.113,E2 -6864.113} C_VEL
LIN {X 0,Y 481.746,Z 431.099,A -85,B 0,C 180,E1 -6867.139,E2 -6867.139} C_VEL
LIN {X 0,Y 481.678,Z 431.113,A -85,B 0,C 180,E1 -6869.741,E2 -6869.741} C_VEL
LIN {X 0,Y 481.672,Z 431.106,A -85,B 0,C 180,E1 -6872.674,E2 -6872.674} C_VEL
LIN {X 0,Y 481.643,Z 431.116,A -85,B 0,C 180,E1 -6875.709,E2 -6875.709} C_VEL
LIN {X 0,Y 481.671,Z 431.107,A -85,B 0,C 180,E1 -6878.859,E2 -6878.859} C_VEL
LIN {X 0,Y 481.652,Z 431.114,A -85,B 0,C 180,E1 -6881.913,E2 -6881.913} C_VEL
LIN {X 0,Y 481.659,Z 431.109,A -85,B 0,C 180,E1 -6884.457,E2 -6884.457} C_VEL
LIN {X 0,Y 481.689,Z 431.105,A -85,B 0,C 180,E1 -6886.846,E2 -6886.846} C_VEL
LIN {X 0,Y 481.677,Z 431.112,A -85,B 0,C 180,E1 -6890.06,E2 -6890.06} C_VEL
LIN {X 0,Y 481.625,Z 431.115,A -85,B 0,C 180,E1 -6893.253,E2 -6893.253} C_VEL
LIN {X 0,Y 481.71,Z 431.108,A -85,B 0,C 180,E1 -6896.33,E2 -6896.33} C_VEL
LIN {X 0,Y 481.692,Z 431.112,A -85,B 0,C 180,E1 -6899.777,E2 -6899.777} C_VEL
LIN {X 0,Y 481.712,Z 431.175,A -85,B 0,C 180,E1 -6900.201,E2 -6900.201} C_VEL
LIN {X 0,Y 485.595,Z 447.41,A -85,B 0,C 180,E1 -6902.877,E2 -6902.877} C_VEL
LIN {X 0,Y 485.952,Z 450.567,A -85,B 0,C 180,E1 -6903.363,E2 -6903.363} C_VEL
LIN {X 0,Y 484.808,Z 472.933,A -85,B 0,C 180,E1 -6906.562,E2 -6906.562} C_VEL
LIN {X 0,Y 488.97,Z 494.998,A -85,B 0,C 180,E1 -6907.143,E2 -6907.143} C_VEL
LIN {X 0,Y 487.461,Z 639.277,A -85,B 0,C 180,E1 -6909.343,E2 -6909.343} C_VEL
LIN {X 0,Y 486.936,Z 655.441,A -85,B 0,C 180,E1 -6909.76,E2 -6909.76} C_VEL
LIN {X 0,Y 486.404,Z 670.341,A -85,B 0,C 180,E1 -6910.324,E2 -6910.324} C_VEL
LIN {X 0,Y 485.735,Z 684.001,A -85,B 0,C 180,E1 -6911.001,E2 -6911.001} C_VEL
LIN {X 0,Y 485.048,Z 697.583,A -85,B 0,C 180,E1 -6911.849,E2 -6911.849} C_VEL
LIN {X 0,Y 484.303,Z 710.094,A -85,B 0,C 180,E1 -6912.802,E2 -6912.802} C_VEL
LIN {X 0,Y 483.549,Z 722.81,A -85,B 0,C 180,E1 -6913.969,E2 -6913.969} C_VEL
LIN {X 0,Y 482.829,Z 734.36,A -85,B 0,C 180,E1 -6915.242,E2 -6915.242} C_VEL
LIN {X 0,Y 482.292,Z 744.084,A -85,B 0,C 180,E1 -6916.517,E2 -6916.517} C_VEL
LIN {X 0,Y 481.762,Z 753.375,A -85,B 0,C 180,E1 -6917.958,E2 -6917.958} C_VEL
LIN {X 0,Y 481.455,Z 761.587,A -85,B 0,C 180,E1 -6919.486,E2 -6919.486} C_VEL
LIN {X 0,Y 481.132,Z 769.011,A -85,B 0,C 180,E1 -6921.177,E2 -6921.177} C_VEL
LIN {X 0,Y 480.986,Z 774.903,A -85,B 0,C 180,E1 -6922.865,E2 -6922.865} C_VEL
LIN {X 0,Y 480.898,Z 778.402,A -85,B 0,C 180,E1 -6924.128,E2 -6924.128} C_VEL
LIN {X 0,Y 480.794,Z 781.939,A -85,B 0,C 180,E1 -6925.808,E2 -6925.808} C_VEL
LIN {X 0,Y 480.798,Z 784.267,A -85,B 0,C 180,E1 -6927.486,E2 -6927.486} C_VEL
LIN {X 0,Y 480.757,Z 785.435,A -85,B 0,C 180,E1 -6929.162,E2 -6929.162} C_VEL
LIN {X 0,Y 480.757,Z 785.43,A -85,B 0,C 180,E1 -6930.837,E2 -6930.837} C_VEL
LIN {X 0,Y 480.798,Z 784.253,A -85,B 0,C 180,E1 -6932.513,E2 -6932.513} C_VEL
LIN {X 0,Y 480.794,Z 781.919,A -85,B 0,C 180,E1 -6934.191,E2 -6934.191} C_VEL
LIN {X 0,Y 480.899,Z 778.381,A -85,B 0,C 180,E1 -6935.871,E2 -6935.871} C_VEL
LIN {X 0,Y 480.993,Z 773.546,A -85,B 0,C 180,E1 -6937.556,E2 -6937.556} C_VEL
LIN {X 0,Y 481.207,Z 767.284,A -85,B 0,C 180,E1 -6939.244,E2 -6939.244} C_VEL
LIN {X 0,Y 481.592,Z 759.424,A -85,B 0,C 180,E1 -6940.935,E2 -6940.935} C_VEL
LIN {X 0,Y 481.857,Z 751.526,A -85,B 0,C 180,E1 -6942.346,E2 -6942.346} C_VEL
LIN {X 0,Y 482.455,Z 740.986,A -85,B 0,C 180,E1 -6943.907,E2 -6943.907} C_VEL
LIN {X 0,Y 483.025,Z 730.689,A -85,B 0,C 180,E1 -6945.182,E2 -6945.182} C_VEL
LIN {X 0,Y 483.768,Z 719.396,A -85,B 0,C 180,E1 -6946.358,E2 -6946.358} C_VEL
LIN {X 0,Y 484.474,Z 706.1,A -85,B 0,C 180,E1 -6947.518,E2 -6947.518} C_VEL
LIN {X 0,Y 485.282,Z 692.696,A -85,B 0,C 180,E1 -6948.469,E2 -6948.469} C_VEL
LIN {X 0,Y 486.008,Z 677.896,A -85,B 0,C 180,E1 -6949.316,E2 -6949.316} C_VEL
LIN {X 0,Y 486.668,Z 662.421,A -85,B 0,C 180,E1 -6949.995,E2 -6949.995} C_VEL
LIN {X 0,Y 487.229,Z 647.184,A -85,B 0,C 180,E1 -6950.474,E2 -6950.474} C_VEL
LIN {X 0,Y 487.542,Z 631.642,A -85,B 0,C 180,E1 -6950.791,E2 -6950.791} C_VEL
LIN {X 0,Y 488.986,Z 495.105,A -85,B 0,C 180,E1 -6952.853,E2 -6952.853} C_VEL
LIN {X 0,Y 484.784,Z 472.681,A -85,B 0,C 180,E1 -6953.444,E2 -6953.444} C_VEL
LIN {X 0,Y 485.896,Z 450.356,A -85,B 0,C 180,E1 -6956.639,E2 -6956.639} C_VEL
LIN {X 0,Y 485.182,Z 445.628,A -85,B 0,C 180,E1 -6957.38,E2 -6957.38} C_VEL
LIN {X 0,Y 481.683,Z 431.114,A -85,B 0,C 180,E1 -6959.8,E2 -6959.8} C_VEL
LIN {X 0,Y 481.67,Z 431.113,A -85,B 0,C 180,E1 -6962.673,E2 -6962.673} C_VEL
LIN {X 0,Y 481.638,Z 431.113,A -85,B 0,C 180,E1 -6965.708,E2 -6965.708} C_VEL
LIN {X 0,Y 481.715,Z 431.102,A -85,B 0,C 180,E1 -6969.354,E2 -6969.354} C_VEL
LIN {X 0,Y 481.669,Z 431.113,A -85,B 0,C 180,E1 -6972.157,E2 -6972.157} C_VEL
LIN {X 0,Y 481.655,Z 431.117,A -85,B 0,C 180,E1 -6974.457,E2 -6974.457} C_VEL
LIN {X 0,Y 481.642,Z 431.112,A -85,B 0,C 180,E1 -6977.839,E2 -6977.839} C_VEL
LIN {X 0,Y 481.674,Z 431.111,A -85,B 0,C 180,E1 -6980.651,E2 -6980.651} C_VEL
LIN {X 0,Y 481.625,Z 431.113,A -85,B 0,C 180,E1 -6983.375,E2 -6983.375} C_VEL
LIN {X 0,Y 481.703,Z 431.109,A -85,B 0,C 180,E1 -6986.33,E2 -6986.33} C_VEL
LIN {X 0,Y 481.644,Z 431.11,A -85,B 0,C 180,E1 -6989.417,E2 -6989.417} C_VEL
LIN {X 0,Y 481.695,Z 431.111,A -85,B 0,C 180,E1 -6992.168,E2 -6992.168} C_VEL
LIN {X 0,Y 481.711,Z 431.103,A -85,B 0,C 180,E1 -6994.97,E2 -6994.97} C_VEL
LIN {X 0,Y 481.645,Z 431.111,A -85,B 0,C 180,E1 -6997.705,E2 -6997.705} C_VEL
LIN {X 0,Y 481.701,Z 431.108,A -85,B 0,C 180,E1 -7000.393,E2 -7000.393} C_VEL
LIN {X 0,Y 481.684,Z 431.103,A -85,B 0,C 180,E1 -7003.034,E2 -7003.034} C_VEL
LIN {X 0,Y 481.682,Z 431.106,A -85,B 0,C 180,E1 -7005.639,E2 -7005.639} C_VEL
LIN {X 0,Y 481.787,Z 431.097,A -85,B 0,C 180,E1 -7008.216,E2 -7008.216} C_VEL
LIN {X 0,Y 481.756,Z 431.096,A -85,B 0,C 180,E1 -7011.612,E2 -7011.612} C_VEL
LIN {X 0,Y 481.809,Z 431.093,A -85,B 0,C 180,E1 -7014.14,E2 -7014.14} C_VEL
LIN {X 0,Y 481.922,Z 431.073,A -85,B 0,C 180,E1 -7017.493,E2 -7017.493} C_VEL
LIN {X 0,Y 481.899,Z 431.077,A -85,B 0,C 180,E1 -7020.836,E2 -7020.836} C_VEL
LIN {X 0,Y 481.922,Z 431.083,A -85,B 0,C 180,E1 -7022.508,E2 -7022.508} C_VEL
LIN {X 0,Y 481.812,Z 431.09,A -85,B 0,C 180,E1 -7025.861,E2 -7025.861} C_VEL
LIN {X 0,Y 481.757,Z 431.101,A -85,B 0,C 180,E1 -7028.389,E2 -7028.389} C_VEL
LIN {X 0,Y 481.743,Z 431.097,A -85,B 0,C 180,E1 -7031.785,E2 -7031.785} C_VEL
LIN {X 0,Y 481.737,Z 431.099,A -85,B 0,C 180,E1 -7035.225,E2 -7035.225} C_VEL
LIN {X 0,Y 481.706,Z 431.106,A -85,B 0,C 180,E1 -7038.722,E2 -7038.722} C_VEL
LIN {X 0,Y 481.641,Z 431.11,A -85,B 0,C 180,E1 -7041.395,E2 -7041.395} C_VEL
LIN {X 0,Y 481.672,Z 431.112,A -85,B 0,C 180,E1 -7044.114,E2 -7044.114} C_VEL
LIN {X 0,Y 481.746,Z 431.1,A -85,B 0,C 180,E1 -7047.141,E2 -7047.141} C_VEL
LIN {X 0,Y 481.683,Z 431.106,A -85,B 0,C 180,E1 -7049.741,E2 -7049.741} C_VEL
LIN {X 0,Y 481.669,Z 431.111,A -85,B 0,C 180,E1 -7052.675,E2 -7052.675} C_VEL
LIN {X 0,Y 481.639,Z 431.114,A -85,B 0,C 180,E1 -7055.71,E2 -7055.71} C_VEL
LIN {X 0,Y 481.716,Z 431.107,A -85,B 0,C 180,E1 -7059.355,E2 -7059.355} C_VEL
LIN {X 0,Y 481.708,Z 431.185,A -85,B 0,C 180,E1 -7061.577,E2 -7061.577} C_VEL
LIN {X 0,Y 484.76,Z 444.829,A -85,B 0,C 180,E1 -7064.099,E2 -7064.099} C_VEL
LIN {X 0,Y 484.889,Z 448.195,A -85,B 0,C 180,E1 -7064.651,E2 -7064.651} C_VEL
LIN {X 0,Y 489.201,Z 467.412,A -85,B 0,C 180,E1 -7065.177,E2 -7065.177} C_VEL
LIN {X 0,Y 487.572,Z 613.114,A -85,B 0,C 180,E1 -7067.403,E2 -7067.403} C_VEL
LIN {X 0,Y 487.332,Z 621.495,A -85,B 0,C 180,E1 -7067.6,E2 -7067.6} C_VEL
LIN {X 0,Y 486.866,Z 625.322,A -85,B 0,C 180,E1 -7067.695,E2 -7067.695} C_VEL
LIN {X 0,Y 485.929,Z 629.102,A -85,B 0,C 180,E1 -7067.773,E2 -7067.773} C_VEL
LIN {X 0,Y 480.941,Z 643.844,A -85,B 0,C 180,E1 -7068.141,E2 -7068.141} C_VEL
LIN {X 0,Y 479.766,Z 649.328,A -85,B 0,C 180,E1 -7068.359,E2 -7068.359} C_VEL
LIN {X 0,Y 479.596,Z 651.145,A -85,B 0,C 180,E1 -7068.446,E2 -7068.446} C_VEL
LIN {X 0,Y 478.892,Z 664.761,A -85,B 0,C 180,E1 -7069.228,E2 -7069.228} C_VEL
LIN {X 0,Y 478.158,Z 677.31,A -85,B 0,C 180,E1 -7070.12,E2 -7070.12} C_VEL
LIN {X 0,Y 477.287,Z 690.317,A -85,B 0,C 180,E1 -7071.237,E2 -7071.237} C_VEL
LIN {X 0,Y 476.528,Z 702.691,A -85,B 0,C 180,E1 -7072.529,E2 -7072.529} C_VEL
LIN {X 0,Y 475.813,Z 712.752,A -85,B 0,C 180,E1 -7073.786,E2 -7073.786} C_VEL
LIN {X 0,Y 475.184,Z 722.872,A -85,B 0,C 180,E1 -7075.291,E2 -7075.291} C_VEL
LIN {X 0,Y 474.726,Z 731.221,A -85,B 0,C 180,E1 -7076.788,E2 -7076.788} C_VEL
LIN {X 0,Y 474.294,Z 739.143,A -85,B 0,C 180,E1 -7078.512,E2 -7078.512} C_VEL
LIN {X 0,Y 474.028,Z 745.408,A -85,B 0,C 180,E1 -7080.221,E2 -7080.221} C_VEL
LIN {X 0,Y 473.835,Z 750.814,A -85,B 0,C 180,E1 -7082.147,E2 -7082.147} C_VEL
LIN {X 0,Y 473.685,Z 753.758,A -85,B 0,C 180,E1 -7083.571,E2 -7083.571} C_VEL
LIN {X 0,Y 473.595,Z 756.369,A -85,B 0,C 180,E1 -7085.449,E2 -7085.449} C_VEL
LIN {X 0,Y 473.582,Z 757.578,A -85,B 0,C 180,E1 -7087.305,E2 -7087.305} C_VEL
LIN {X 0,Y 473.608,Z 757.417,A -85,B 0,C 180,E1 -7089.209,E2 -7089.209} C_VEL
LIN {X 0,Y 473.628,Z 756.054,A -85,B 0,C 180,E1 -7090.947,E2 -7090.947} C_VEL
LIN {X 0,Y 473.719,Z 753.362,A -85,B 0,C 180,E1 -7092.74,E2 -7092.74} C_VEL
LIN {X 0,Y 473.92,Z 749.241,A -85,B 0,C 180,E1 -7094.563,E2 -7094.563} C_VEL
LIN {X 0,Y 474.077,Z 744.007,A -85,B 0,C 180,E1 -7096.28,E2 -7096.28} C_VEL
LIN {X 0,Y 474.421,Z 737.19,A -85,B 0,C 180,E1 -7098.031,E2 -7098.031} C_VEL
LIN {X 0,Y 474.847,Z 728.745,A -85,B 0,C 180,E1 -7099.77,E2 -7099.77} C_VEL
LIN {X 0,Y 475.394,Z 719.743,A -85,B 0,C 180,E1 -7101.285,E2 -7101.285} C_VEL
LIN {X 0,Y 476.079,Z 708.972,A -85,B 0,C 180,E1 -7102.792,E2 -7102.792} C_VEL
LIN {X 0,Y 476.903,Z 696.878,A -85,B 0,C 180,E1 -7104.186,E2 -7104.186} C_VEL
LIN {X 0,Y 477.627,Z 684.646,A -85,B 0,C 180,E1 -7105.359,E2 -7105.359} C_VEL
LIN {X 0,Y 478.484,Z 671.125,A -85,B 0,C 180,E1 -7106.422,E2 -7106.422} C_VEL
LIN {X 0,Y 479.244,Z 657.366,A -85,B 0,C 180,E1 -7107.299,E2 -7107.299} C_VEL
LIN {X 0,Y 479.946,Z 643.309,A -85,B 0,C 180,E1 -7108.007,E2 -7108.007} C_VEL
LIN {X 0,Y 480.493,Z 628.147,A -85,B 0,C 180,E1 -7108.586,E2 -7108.586} C_VEL
LIN {X 0,Y 480.916,Z 613.215,A -85,B 0,C 180,E1 -7108.98,E2 -7108.98} C_VEL
LIN {X 0,Y 482.546,Z 467.673,A -85,B 0,C 180,E1 -7111.237,E2 -7111.237} C_VEL
LIN {X 0,Y 478.023,Z 447.822,A -85,B 0,C 180,E1 -7111.813,E2 -7111.813} C_VEL
LIN {X 0,Y 476.706,Z 440.358,A -85,B 0,C 180,E1 -7113.17,E2 -7113.17} C_VEL
LIN {X 0,Y 474.689,Z 431.98,A -85,B 0,C 180,E1 -7114.778,E2 -7114.778} C_VEL
LIN {X 0,Y 474.734,Z 431.977,A -85,B 0,C 180,E1 -7117.307,E2 -7117.307} C_VEL
LIN {X 0,Y 474.687,Z 431.974,A -85,B 0,C 180,E1 -7120.234,E2 -7120.234} C_VEL
LIN {X 0,Y 474.683,Z 431.981,A -85,B 0,C 180,E1 -7122.832,E2 -7122.832} C_VEL
LIN {X 0,Y 474.685,Z 431.982,A -85,B 0,C 180,E1 -7125.768,E2 -7125.768} C_VEL
LIN {X 0,Y 474.669,Z 431.981,A -85,B 0,C 180,E1 -7129.01,E2 -7129.01} C_VEL
LIN {X 0,Y 474.596,Z 431.994,A -85,B 0,C 180,E1 -7131.729,E2 -7131.729} C_VEL
LIN {X 0,Y 474.664,Z 431.977,A -85,B 0,C 180,E1 -7134.493,E2 -7134.493} C_VEL
LIN {X 0,Y 474.703,Z 431.979,A -85,B 0,C 180,E1 -7137.339,E2 -7137.339} C_VEL
LIN {X 0,Y 474.609,Z 431.987,A -85,B 0,C 180,E1 -7140.81,E2 -7140.81} C_VEL
LIN {X 0,Y 474.642,Z 431.987,A -85,B 0,C 180,E1 -7143.984,E2 -7143.984} C_VEL
LIN {X 0,Y 474.578,Z 431.989,A -85,B 0,C 180,E1 -7146.9,E2 -7146.9} C_VEL
LIN {X 0,Y 474.631,Z 431.988,A -85,B 0,C 180,E1 -7149.648,E2 -7149.648} C_VEL
LIN {X 0,Y 474.638,Z 431.981,A -85,B 0,C 180,E1 -7152.932,E2 -7152.932} C_VEL
LIN {X 0,Y 474.612,Z 431.991,A -85,B 0,C 180,E1 -7155.895,E2 -7155.895} C_VEL
LIN {X 0,Y 474.643,Z 431.978,A -85,B 0,C 180,E1 -7159.039,E2 -7159.039} C_VEL
LIN {X 0,Y 474.619,Z 431.992,A -85,B 0,C 180,E1 -7161.703,E2 -7161.703} C_VEL
LIN {X 0,Y 474.632,Z 431.979,A -85,B 0,C 180,E1 -7164.726,E2 -7164.726} C_VEL
LIN {X 0,Y 474.637,Z 431.988,A -85,B 0,C 180,E1 -7167.788,E2 -7167.788} C_VEL
LIN {X 0,Y 474.625,Z 431.979,A -85,B 0,C 180,E1 -7170.884,E2 -7170.884} C_VEL
LIN {X 0,Y 474.669,Z 431.987,A -85,B 0,C 180,E1 -7173.629,E2 -7173.629} C_VEL
LIN {X 0,Y 474.636,Z 431.974,A -85,B 0,C 180,E1 -7176.641,E2 -7176.641} C_VEL
LIN {X 0,Y 474.655,Z 431.983,A -85,B 0,C 180,E1 -7180.089,E2 -7180.089} C_VEL
LIN {X 0,Y 474.651,Z 431.975,A -85,B 0,C 180,E1 -7182.774,E2 -7182.774} C_VEL
LIN {X 0,Y 474.648,Z 431.982,A -85,B 0,C 180,E1 -7185.421,E2 -7185.421} C_VEL
LIN {X 0,Y 474.704,Z 431.975,A -85,B 0,C 180,E1 -7188.037,E2 -7188.037} C_VEL
LIN {X 0,Y 474.728,Z 431.97,A -85,B 0,C 180,E1 -7191.486,E2 -7191.486} C_VEL
LIN {X 0,Y 474.779,Z 431.968,A -85,B 0,C 180,E1 -7194.052,E2 -7194.052} C_VEL
LIN {X 0,Y 474.894,Z 431.948,A -85,B 0,C 180,E1 -7197.455,E2 -7197.455} C_VEL
LIN {X 0,Y 474.911,Z 431.953,A -85,B 0,C 180,E1 -7200,E2 -7200} C_VEL
LIN {X 0,Y 474.894,Z 431.947,A -85,B 0,C 180,E1 -7202.544,E2 -7202.544} C_VEL
LIN {X 0,Y 474.778,Z 431.968,A -85,B 0,C 180,E1 -7205.947,E2 -7205.947} C_VEL
LIN {X 0,Y 474.728,Z 431.972,A -85,B 0,C 180,E1 -7208.513,E2 -7208.513} C_VEL
LIN {X 0,Y 474.703,Z 431.971,A -85,B 0,C 180,E1 -7211.962,E2 -7211.962} C_VEL
LIN {X 0,Y 474.699,Z 431.98,A -85,B 0,C 180,E1 -7215.455,E2 -7215.455} C_VEL
LIN {X 0,Y 474.664,Z 431.972,A -85,B 0,C 180,E1 -7219.01,E2 -7219.01} C_VEL
LIN {X 0,Y 474.589,Z 431.996,A -85,B 0,C 180,E1 -7221.729,E2 -7221.729} C_VEL
LIN {X 0,Y 474.658,Z 431.981,A -85,B 0,C 180,E1 -7224.493,E2 -7224.493} C_VEL
LIN {X 0,Y 474.699,Z 431.979,A -85,B 0,C 180,E1 -7227.339,E2 -7227.339} C_VEL
LIN {X 0,Y 474.603,Z 431.986,A -85,B 0,C 180,E1 -7230.81,E2 -7230.81} C_VEL
LIN {X 0,Y 474.638,Z 431.988,A -85,B 0,C 180,E1 -7233.984,E2 -7233.984} C_VEL
LIN {X 0,Y 474.575,Z 431.991,A -85,B 0,C 180,E1 -7236.9,E2 -7236.9} C_VEL
LIN {X 0,Y 474.627,Z 431.992,A -85,B 0,C 180,E1 -7239.648,E2 -7239.648} C_VEL
LIN {X 0,Y 474.614,Z 431.986,A -85,B 0,C 180,E1 -7242.934,E2 -7242.934} C_VEL
LIN {X 0,Y 474.618,Z 431.991,A -85,B 0,C 180,E1 -7245.896,E2 -7245.896} C_VEL
LIN {X 0,Y 474.632,Z 431.986,A -85,B 0,C 180,E1 -7249.04,E2 -7249.04} C_VEL
LIN {X 0,Y 474.61,Z 431.994,A -85,B 0,C 180,E1 -7251.704,E2 -7251.704} C_VEL
LIN {X 0,Y 474.624,Z 431.989,A -85,B 0,C 180,E1 -7254.726,E2 -7254.726} C_VEL
LIN {X 0,Y 474.636,Z 431.987,A -85,B 0,C 180,E1 -7257.788,E2 -7257.788} C_VEL
LIN {X 0,Y 474.673,Z 432.132,A -85,B 0,C 180,E1 -7259.897,E2 -7259.897} C_VEL
LIN {X 0,Y 478.685,Z 448.815,A -85,B 0,C 180,E1 -7262.696,E2 -7262.696} C_VEL
LIN {X 0,Y 479.098,Z 452.95,A -85,B 0,C 180,E1 -7263.339,E2 -7263.339} C_VEL
LIN {X 0,Y 478.034,Z 473.149,A -85,B 0,C 180,E1 -7266.244,E2 -7266.244} C_VEL
LIN {X 0,Y 482.401,Z 496.126,A -85,B 0,C 180,E1 -7266.836,E2 -7266.836} C_VEL
LIN {X 0,Y 480.806,Z 638.882,A -85,B 0,C 180,E1 -7269.043,E2 -7269.043} C_VEL
LIN {X 0,Y 480.307,Z 654.829,A -85,B 0,C 180,E1 -7269.457,E2 -7269.457} C_VEL
LIN {X 0,Y 479.681,Z 670.44,A -85,B 0,C 180,E1 -7270.055,E2 -7270.055} C_VEL
LIN {X 0,Y 478.986,Z 683.737,A -85,B 0,C 180,E1 -7270.723,E2 -7270.723} C_VEL
LIN {X 0,Y 478.236,Z 697.333,A -85,B 0,C 180,E1 -7271.581,E2 -7271.581} C_VEL
LIN {X 0,Y 477.479,Z 709.857,A -85,B 0,C 180,E1 -7272.548,E2 -7272.548} C_VEL
LIN {X 0,Y 476.674,Z 722.583,A -85,B 0,C 180,E1 -7273.732,E2 -7273.732} C_VEL
LIN {X 0,Y 475.889,Z 734.139,A -85,B 0,C 180,E1 -7275.022,E2 -7275.022} C_VEL
LIN {X 0,Y 475.33,Z 743.867,A -85,B 0,C 180,E1 -7276.316,E2 -7276.316} C_VEL
LIN {X 0,Y 474.712,Z 752.828,A -85,B 0,C 180,E1 -7277.718,E2 -7277.718} C_VEL
LIN {X 0,Y 474.412,Z 761.375,A -85,B 0,C 180,E1 -7279.328,E2 -7279.328} C_VEL
LIN {X 0,Y 474.08,Z 768.802,A -85,B 0,C 180,E1 -7281.045,E2 -7281.045} C_VEL
LIN {X 0,Y 473.907,Z 774.694,A -85,B 0,C 180,E1 -7282.758,E2 -7282.758} C_VEL
LIN {X 0,Y 473.806,Z 778.194,A -85,B 0,C 180,E1 -7284.04,E2 -7284.04} C_VEL
LIN {X 0,Y 473.703,Z 781.732,A -85,B 0,C 180,E1 -7285.745,E2 -7285.745} C_VEL
LIN {X 0,Y 473.717,Z 784.06,A -85,B 0,C 180,E1 -7287.449,E2 -7287.449} C_VEL
LIN {X 0,Y 473.685,Z 785.229,A -85,B 0,C 180,E1 -7289.149,E2 -7289.149} C_VEL
LIN {X 0,Y 473.685,Z 785.223,A -85,B 0,C 180,E1 -7290.85,E2 -7290.85} C_VEL
LIN {X 0,Y 473.718,Z 784.044,A -85,B 0,C 180,E1 -7292.55,E2 -7292.55} C_VEL
LIN {X 0,Y 473.703,Z 781.708,A -85,B 0,C 180,E1 -7294.254,E2 -7294.254} C_VEL
LIN {X 0,Y 473.81,Z 778.168,A -85,B 0,C 180,E1 -7295.959,E2 -7295.959} C_VEL
LIN {X 0,Y 473.915,Z 773.329,A -85,B 0,C 180,E1 -7297.669,E2 -7297.669} C_VEL
LIN {X 0,Y 474.137,Z 767.065,A -85,B 0,C 180,E1 -7299.383,E2 -7299.383} C_VEL
LIN {X 0,Y 474.567,Z 759.201,A -85,B 0,C 180,E1 -7301.099,E2 -7301.099} C_VEL
LIN {X 0,Y 474.914,Z 750.564,A -85,B 0,C 180,E1 -7302.65,E2 -7302.65} C_VEL
LIN {X 0,Y 475.47,Z 740.756,A -85,B 0,C 180,E1 -7304.116,E2 -7304.116} C_VEL
LIN {X 0,Y 476.097,Z 730.459,A -85,B 0,C 180,E1 -7305.409,E2 -7305.409} C_VEL
LIN {X 0,Y 476.937,Z 718.16,A -85,B 0,C 180,E1 -7306.701,E2 -7306.701} C_VEL
LIN {X 0,Y 477.655,Z 705.867,A -85,B 0,C 180,E1 -7307.776,E2 -7307.776} C_VEL
LIN {X 0,Y 478.481,Z 692.459,A -85,B 0,C 180,E1 -7308.741,E2 -7308.741} C_VEL
LIN {X 0,Y 479.296,Z 677.655,A -85,B 0,C 180,E1 -7309.597,E2 -7309.597} C_VEL
LIN {X 0,Y 479.934,Z 663.089,A -85,B 0,C 180,E1 -7310.249,E2 -7310.249} C_VEL
LIN {X 0,Y 480.513,Z 647.865,A -85,B 0,C 180,E1 -7310.745,E2 -7310.745} C_VEL
LIN {X 0,Y 480.891,Z 632.898,A -85,B 0,C 180,E1 -7311.064,E2 -7311.064} C_VEL
LIN {X 0,Y 482.435,Z 496.262,A -85,B 0,C 180,E1 -7313.161,E2 -7313.161} C_VEL
LIN {X 0,Y 477.96,Z 472.576,A -85,B 0,C 180,E1 -7313.784,E2 -7313.784} C_VEL
LIN {X 0,Y 479.067,Z 451.354,A -85,B 0,C 180,E1 -7316.872,E2 -7316.872} C_VEL
LIN {X 0,Y 476.792,Z 440.699,A -85,B 0,C 180,E1 -7318.623,E2 -7318.623} C_VEL
LIN {X 0,Y 474.653,Z 431.989,A -85,B 0,C 180,E1 -7320.134,E2 -7320.134} C_VEL
LIN {X 0,Y 474.639,Z 431.986,A -85,B 0,C 180,E1 -7323.219,E2 -7323.219} C_VEL
LIN {X 0,Y 474.589,Z 431.998,A -85,B 0,C 180,E1 -7326.322,E2 -7326.322} C_VEL
LIN {X 0,Y 474.651,Z 431.984,A -85,B 0,C 180,E1 -7329.651,E2 -7329.651} C_VEL
LIN {X 0,Y 474.647,Z 431.981,A -85,B 0,C 180,E1 -7332.929,E2 -7332.929} C_VEL
LIN {X 0,Y 474.603,Z 431.993,A -85,B 0,C 180,E1 -7335.895,E2 -7335.895} C_VEL
LIN {X 0,Y 474.622,Z 431.987,A -85,B 0,C 180,E1 -7339.04,E2 -7339.04} C_VEL
LIN {X 0,Y 474.604,Z 431.99,A -85,B 0,C 180,E1 -7341.703,E2 -7341.703} C_VEL
LIN {X 0,Y 474.624,Z 431.988,A -85,B 0,C 180,E1 -7344.726,E2 -7344.726} C_VEL
LIN {X 0,Y 474.631,Z 431.984,A -85,B 0,C 180,E1 -7347.788,E2 -7347.788} C_VEL
LIN {X 0,Y 474.617,Z 431.988,A -85,B 0,C 180,E1 -7350.884,E2 -7350.884} C_VEL
LIN {X 0,Y 474.659,Z 431.979,A -85,B 0,C 180,E1 -7353.629,E2 -7353.629} C_VEL
LIN {X 0,Y 474.628,Z 431.989,A -85,B 0,C 180,E1 -7356.641,E2 -7356.641} C_VEL
LIN {X 0,Y 474.649,Z 431.983,A -85,B 0,C 180,E1 -7360.09,E2 -7360.09} C_VEL
LIN {X 0,Y 474.644,Z 431.982,A -85,B 0,C 180,E1 -7362.774,E2 -7362.774} C_VEL
LIN {X 0,Y 474.64,Z 431.983,A -85,B 0,C 180,E1 -7365.421,E2 -7365.421} C_VEL
LIN {X 0,Y 474.731,Z 431.974,A -85,B 0,C 180,E1 -7368.038,E2 -7368.038} C_VEL
LIN {X 0,Y 474.721,Z 431.972,A -85,B 0,C 180,E1 -7371.487,E2 -7371.487} C_VEL
LIN {X 0,Y 474.772,Z 431.969,A -85,B 0,C 180,E1 -7374.053,E2 -7374.053} C_VEL
LIN {X 0,Y 474.888,Z 431.95,A -85,B 0,C 180,E1 -7377.456,E2 -7377.456} C_VEL
LIN {X 0,Y 474.85,Z 431.955,A -85,B 0,C 180,E1 -7380.848,E2 -7380.848} C_VEL
LIN {X 0,Y 474.888,Z 431.958,A -85,B 0,C 180,E1 -7382.545,E2 -7382.545} C_VEL
LIN {X 0,Y 474.774,Z 431.968,A -85,B 0,C 180,E1 -7385.948,E2 -7385.948} C_VEL
LIN {X 0,Y 474.722,Z 431.978,A -85,B 0,C 180,E1 -7388.514,E2 -7388.514} C_VEL
LIN {X 0,Y 474.697,Z 431.977,A -85,B 0,C 180,E1 -7391.963,E2 -7391.963} C_VEL
LIN {X 0,Y 474.694,Z 431.977,A -85,B 0,C 180,E1 -7395.456,E2 -7395.456} C_VEL
LIN {X 0,Y 474.659,Z 431.982,A -85,B 0,C 180,E1 -7399.011,E2 -7399.011} C_VEL
LIN {X 0,Y 474.584,Z 431.991,A -85,B 0,C 180,E1 -7401.729,E2 -7401.729} C_VEL
LIN {X 0,Y 474.653,Z 431.991,A -85,B 0,C 180,E1 -7404.493,E2 -7404.493} C_VEL
LIN {X 0,Y 474.693,Z 431.978,A -85,B 0,C 180,E1 -7407.339,E2 -7407.339} C_VEL
LIN {X 0,Y 474.605,Z 431.993,A -85,B 0,C 180,E1 -7410.812,E2 -7410.812} C_VEL
LIN {X 0,Y 474.634,Z 431.988,A -85,B 0,C 180,E1 -7413.985,E2 -7413.985} C_VEL
LIN {X 0,Y 474.572,Z 431.996,A -85,B 0,C 180,E1 -7416.901,E2 -7416.901} C_VEL
LIN {X 0,Y 474.651,Z 431.987,A -85,B 0,C 180,E1 -7419.652,E2 -7419.652} C_VEL
LIN {X 0,Y 474.677,Z 432.119,A -85,B 0,C 180,E1 -7421.276,E2 -7421.276} C_VEL
LIN {X 0,Y 477.788,Z 445.983,A -85,B 0,C 180,E1 -7423.884,E2 -7423.884} C_VEL
LIN {X 0,Y 478.058,Z 448.271,A -85,B 0,C 180,E1 -7424.291,E2 -7424.291} C_VEL
LIN {X 0,Y 482.688,Z 468.069,A -85,B 0,C 180,E1 -7424.856,E2 -7424.856} C_VEL
LIN {X 0,Y 480.935,Z 613.666,A -85,B 0,C 180,E1 -7427.114,E2 -7427.114} C_VEL
LIN {X 0,Y 480.447,Z 629.291,A -85,B 0,C 180,E1 -7427.532,E2 -7427.532} C_VEL
LIN {X 0,Y 479.953,Z 643.434,A -85,B 0,C 180,E1 -7428.078,E2 -7428.078} C_VEL
LIN {X 0,Y 479.596,Z 651.145,A -85,B 0,C 180,E1 -7428.446,E2 -7428.446} C_VEL
LIN {X 0,Y 478.653,Z 656.581,A -85,B 0,C 180,E1 -7428.707,E2 -7428.707} C_VEL
LIN {X 0,Y 475.399,Z 665.345,A -85,B 0,C 180,E1 -7429.117,E2 -7429.117} C_VEL
LIN {X 0,Y 472.192,Z 673.841,A -85,B 0,C 180,E1 -7429.594,E2 -7429.594} C_VEL
LIN {X 0,Y 471.315,Z 678.799,A -85,B 0,C 180,E1 -7429.955,E2 -7429.955} C_VEL
LIN {X 0,Y 470.378,Z 692.058,A -85,B 0,C 180,E1 -7431.133,E2 -7431.133} C_VEL
LIN {X 0,Y 469.603,Z 703.582,A -85,B 0,C 180,E1 -7432.374,E2 -7432.374} C_VEL
LIN {X 0,Y 468.846,Z 713.697,A -85,B 0,C 180,E1 -7433.67,E2 -7433.67} C_VEL
LIN {X 0,Y 468.162,Z 723.827,A -85,B 0,C 180,E1 -7435.219,E2 -7435.219} C_VEL
LIN {X 0,Y 467.71,Z 732.05,A -85,B 0,C 180,E1 -7436.739,E2 -7436.739} C_VEL
LIN {X 0,Y 467.266,Z 738.817,A -85,B 0,C 180,E1 -7438.237,E2 -7438.237} C_VEL
LIN {X 0,Y 467.042,Z 744.405,A -85,B 0,C 180,E1 -7439.729,E2 -7439.729} C_VEL
LIN {X 0,Y 466.829,Z 748.876,A -85,B 0,C 180,E1 -7441.201,E2 -7441.201} C_VEL
LIN {X 0,Y 466.713,Z 752.386,A -85,B 0,C 180,E1 -7442.68,E2 -7442.68} C_VEL
LIN {X 0,Y 466.535,Z 755.723,A -85,B 0,C 180,E1 -7444.67,E2 -7444.67} C_VEL
LIN {X 0,Y 466.486,Z 757.115,A -85,B 0,C 180,E1 -7445.998,E2 -7445.998} C_VEL
LIN {X 0,Y 466.474,Z 757.89,A -85,B 0,C 180,E1 -7447.874,E2 -7447.874} C_VEL
LIN {X 0,Y 466.529,Z 757.345,A -85,B 0,C 180,E1 -7449.728,E2 -7449.728} C_VEL
LIN {X 0,Y 466.594,Z 755.459,A -85,B 0,C 180,E1 -7451.61,E2 -7451.61} C_VEL
LIN {X 0,Y 466.695,Z 752.426,A -85,B 0,C 180,E1 -7453.375,E2 -7453.375} C_VEL
LIN {X 0,Y 466.911,Z 748.012,A -85,B 0,C 180,E1 -7455.175,E2 -7455.175} C_VEL
LIN {X 0,Y 467.081,Z 742.239,A -85,B 0,C 180,E1 -7456.957,E2 -7456.957} C_VEL
LIN {X 0,Y 467.514,Z 734.922,A -85,B 0,C 180,E1 -7458.731,E2 -7458.731} C_VEL
LIN {X 0,Y 467.918,Z 727.138,A -85,B 0,C 180,E1 -7460.273,E2 -7460.273} C_VEL
LIN {X 0,Y 468.503,Z 718.433,A -85,B 0,C 180,E1 -7461.713,E2 -7461.713} C_VEL
LIN {X 0,Y 469.223,Z 708.315,A -85,B 0,C 180,E1 -7463.119,E2 -7463.119} C_VEL
LIN {X 0,Y 470.045,Z 697.088,A -85,B 0,C 180,E1 -7464.423,E2 -7464.423} C_VEL
LIN {X 0,Y 470.84,Z 684.839,A -85,B 0,C 180,E1 -7465.613,E2 -7465.613} C_VEL
LIN {X 0,Y 471.689,Z 672.033,A -85,B 0,C 180,E1 -7466.641,E2 -7466.641} C_VEL
LIN {X 0,Y 472.502,Z 658.106,A -85,B 0,C 180,E1 -7467.55,E2 -7467.55} C_VEL
LIN {X 0,Y 473.258,Z 643.502,A -85,B 0,C 180,E1 -7468.299,E2 -7468.299} C_VEL
LIN {X 0,Y 473.845,Z 628.316,A -85,B 0,C 180,E1 -7468.885,E2 -7468.885} C_VEL
